LIN {X 0,Y 474.699,Z 220.358,A -85,B 0,C 180,E1 -7395.456,E2 -7395.456} C_VEL
LIN {X 0,Y 474.663,Z 220.354,A -85,B 0,C 180,E1 -7399.011,E2 -7399.011} C_VEL
LIN {X 0,Y 474.589,Z 220.363,A -85,B 0,C 180,E1 -7401.729,E2 -7401.729} C_VEL
LIN {X 0,Y 474.629,Z 220.358,A -85,B 0,C 180,E1 -7404.495,E2 -7404.495} C_VEL
LIN {X 0,Y 474.675,Z 220.357,A -85,B 0,C 180,E1 -7407.333,E2 -7407.333} C_VEL
LIN {X 0,Y 474.605,Z 220.36,A -85,B 0,C 180,E1 -7410.23,E2 -7410.23} C_VEL
LIN {X 0,Y 474.645,Z 220.363,A -85,B 0,C 180,E1 -7413.22,E2 -7413.22} C_VEL
LIN {X 0,Y 474.586,Z 220.363,A -85,B 0,C 180,E1 -7416.324,E2 -7416.324} C_VEL
LIN {X 0,Y 474.615,Z 220.366,A -85,B 0,C 180,E1 -7419.646,E2 -7419.646} C_VEL
LIN {X 0,Y 474.602,Z 220.363,A -85,B 0,C 180,E1 -7422.234,E2 -7422.234} C_VEL
LIN {X 0,Y 474.618,Z 220.369,A -85,B 0,C 180,E1 -7425.298,E2 -7425.298} C_VEL
LIN {X 0,Y 474.617,Z 220.364,A -85,B 0,C 180,E1 -7428.214,E2 -7428.214} C_VEL
LIN {X 0,Y 474.612,Z 220.371,A -85,B 0,C 180,E1 -7431.543,E2 -7431.543} C_VEL
LIN {X 0,Y 474.624,Z 220.364,A -85,B 0,C 180,E1 -7434.726,E2 -7434.726} C_VEL
LIN {X 0,Y 474.638,Z 220.362,A -85,B 0,C 180,E1 -7437.788,E2 -7437.788} C_VEL
LIN {X 0,Y 474.61,Z 220.362,A -85,B 0,C 180,E1 -7440.889,E2 -7440.889} C_VEL
LIN {X 0,Y 474.677,Z 220.486,A -85,B 0,C 180,E1 -7442.491,E2 -7442.491} C_VEL
LIN {X 0,Y 475.888,Z 227.892,A -85,B 0,C 180,E1 -7444.05,E2 -7444.05} C_VEL
LIN {X 0,Y 475.509,Z 242.561,A -85,B 0,C 180,E1 -7446.942,E2 -7446.942} C_VEL
LIN {X 0,Y 475.457,Z 243.986,A -85,B 0,C 180,E1 -7447.219,E2 -7447.219} C_VEL
LIN {X 0,Y 477.495,Z 254.111,A -85,B 0,C 180,E1 -7447.465,E2 -7447.465} C_VEL
LIN {X 0,Y 477.669,Z 257.985,A -85,B 0,C 180,E1 -7447.532,E2 -7447.532} C_VEL
LIN {X 0,Y 477.181,Z 261.87,A -85,B 0,C 180,E1 -7447.573,E2 -7447.573} C_VEL
LIN {X 0,Y 475.045,Z 269.533,A -85,B 0,C 180,E1 -7447.609,E2 -7447.609} C_VEL
LIN {X 0,Y 472.115,Z 279.174,A -85,B 0,C 180,E1 -7447.645,E2 -7447.645} C_VEL
LIN {X 0,Y 471.398,Z 285.1,A -85,B 0,C 180,E1 -7447.71,E2 -7447.71} C_VEL
LIN {X 0,Y 470.736,Z 351.494,A -85,B 0,C 180,E1 -7448.745,E2 -7448.745} C_VEL
LIN {X 0,Y 470.477,Z 364.16,A -85,B 0,C 180,E1 -7449.106,E2 -7449.106} C_VEL
LIN {X 0,Y 470.075,Z 377.21,A -85,B 0,C 180,E1 -7449.659,E2 -7449.659} C_VEL
LIN {X 0,Y 469.661,Z 388.302,A -85,B 0,C 180,E1 -7450.296,E2 -7450.296} C_VEL
LIN {X 0,Y 469.132,Z 400.52,A -85,B 0,C 180,E1 -7451.211,E2 -7451.211} C_VEL
LIN {X 0,Y 468.614,Z 411.084,A -85,B 0,C 180,E1 -7452.207,E2 -7452.207} C_VEL
LIN {X 0,Y 468.122,Z 419.679,A -85,B 0,C 180,E1 -7453.202,E2 -7453.202} C_VEL
LIN {X 0,Y 467.705,Z 427.565,A -85,B 0,C 180,E1 -7454.307,E2 -7454.307} C_VEL
LIN {X 0,Y 467.365,Z 435.229,A -85,B 0,C 180,E1 -7455.634,E2 -7455.634} C_VEL
LIN {X 0,Y 467.136,Z 441.363,A -85,B 0,C 180,E1 -7456.958,E2 -7456.958} C_VEL
LIN {X 0,Y 466.936,Z 446.542,A -85,B 0,C 180,E1 -7458.382,E2 -7458.382} C_VEL
LIN {X 0,Y 466.762,Z 449.893,A -85,B 0,C 180,E1 -7459.59,E2 -7459.59} C_VEL
LIN {X 0,Y 466.642,Z 451.795,A -85,B 0,C 180,E1 -7460.464,E2 -7460.464} C_VEL
LIN {X 0,Y 466.643,Z 453.238,A -85,B 0,C 180,E1 -7461.338,E2 -7461.338} C_VEL
LIN {X 0,Y 466.676,Z 454.878,A -85,B 0,C 180,E1 -7463.08,E2 -7463.08} C_VEL
LIN {X 0,Y 466.646,Z 455.12,A -85,B 0,C 180,E1 -7463.948,E2 -7463.948} C_VEL
LIN {X 0,Y 466.65,Z 454.939,A -85,B 0,C 180,E1 -7464.815,E2 -7464.815} C_VEL
LIN {X 0,Y 466.683,Z 453.385,A -85,B 0,C 180,E1 -7466.547,E2 -7466.547} C_VEL
LIN {X 0,Y 466.706,Z 452.028,A -85,B 0,C 180,E1 -7467.411,E2 -7467.411} C_VEL
LIN {X 0,Y 466.724,Z 449.165,A -85,B 0,C 180,E1 -7468.706,E2 -7468.706} C_VEL
LIN {X 0,Y 466.769,Z 445.291,A -85,B 0,C 180,E1 -7470,E2 -7470} C_VEL
LIN {X 0,Y 467.063,Z 440.289,A -85,B 0,C 180,E1 -7471.293,E2 -7471.293} C_VEL
LIN {X 0,Y 467.253,Z 434.025,A -85,B 0,C 180,E1 -7472.586,E2 -7472.586} C_VEL
LIN {X 0,Y 467.656,Z 426.185,A -85,B 0,C 180,E1 -7473.878,E2 -7473.878} C_VEL
LIN {X 0,Y 468.117,Z 418.205,A -85,B 0,C 180,E1 -7474.952,E2 -7474.952} C_VEL
LIN {X 0,Y 468.566,Z 408.492,A -85,B 0,C 180,E1 -7476.027,E2 -7476.027} C_VEL
LIN {X 0,Y 469.086,Z 397.645,A -85,B 0,C 180,E1 -7476.992,E2 -7476.992} C_VEL
LIN {X 0,Y 469.593,Z 385.29,A -85,B 0,C 180,E1 -7477.849,E2 -7477.849} C_VEL
LIN {X 0,Y 470.024,Z 373.161,A -85,B 0,C 180,E1 -7478.491,E2 -7478.491} C_VEL
LIN {X 0,Y 470.342,Z 360.402,A -85,B 0,C 180,E1 -7478.972,E2 -7478.972} C_VEL
LIN {X 0,Y 470.527,Z 346.91,A -85,B 0,C 180,E1 -7479.294,E2 -7479.294} C_VEL
LIN {X 0,Y 471.18,Z 259.024,A -85,B 0,C 180,E1 -7480.637,E2 -7480.637} C_VEL
LIN {X 0,Y 468.414,Z 244.125,A -85,B 0,C 180,E1 -7480.974,E2 -7480.974} C_VEL
LIN {X 0,Y 468.806,Z 229.463,A -85,B 0,C 180,E1 -7483.878,E2 -7483.878} C_VEL
LIN {X 0,Y 468.381,Z 225.11,A -85,B 0,C 180,E1 -7484.778,E2 -7484.778} C_VEL
LIN {X 0,Y 467.657,Z 221.233,A -85,B 0,C 180,E1 -7485.638,E2 -7485.638} C_VEL
LIN {X 0,Y 467.617,Z 221.24,A -85,B 0,C 180,E1 -7488.763,E2 -7488.763} C_VEL
LIN {X 0,Y 467.584,Z 221.237,A -85,B 0,C 180,E1 -7491.268,E2 -7491.268} C_VEL
LIN {X 0,Y 467.566,Z 221.238,A -85,B 0,C 180,E1 -7493.944,E2 -7493.944} C_VEL
LIN {X 0,Y 467.568,Z 221.245,A -85,B 0,C 180,E1 -7496.803,E2 -7496.803} C_VEL
LIN {X 0,Y 467.55,Z 221.24,A -85,B 0,C 180,E1 -7499.738,E2 -7499.738} C_VEL
LIN {X 0,Y 467.586,Z 221.243,A -85,B 0,C 180,E1 -7502.758,E2 -7502.758} C_VEL
LIN {X 0,Y 467.555,Z 221.24,A -85,B 0,C 180,E1 -7505.889,E2 -7505.889} C_VEL
LIN {X 0,Y 467.577,Z 221.239,A -85,B 0,C 180,E1 -7509.145,E2 -7509.145} C_VEL
LIN {X 0,Y 467.588,Z 221.242,A -85,B 0,C 180,E1 -7512.567,E2 -7512.567} C_VEL
LIN {X 0,Y 467.567,Z 221.241,A -85,B 0,C 180,E1 -7515.052,E2 -7515.052} C_VEL
LIN {X 0,Y 467.575,Z 221.245,A -85,B 0,C 180,E1 -7518.596,E2 -7518.596} C_VEL
LIN {X 0,Y 467.56,Z 221.239,A -85,B 0,C 180,E1 -7521.409,E2 -7521.409} C_VEL
LIN {X 0,Y 467.559,Z 221.242,A -85,B 0,C 180,E1 -7524.261,E2 -7524.261} C_VEL
LIN {X 0,Y 467.583,Z 221.237,A -85,B 0,C 180,E1 -7527.321,E2 -7527.321} C_VEL
LIN {X 0,Y 467.57,Z 221.246,A -85,B 0,C 180,E1 -7530.667,E2 -7530.667} C_VEL
LIN {X 0,Y 467.587,Z 221.237,A -85,B 0,C 180,E1 -7533.198,E2 -7533.198} C_VEL
LIN {X 0,Y 467.59,Z 221.241,A -85,B 0,C 180,E1 -7536.469,E2 -7536.469} C_VEL
LIN {X 0,Y 467.623,Z 221.231,A -85,B 0,C 180,E1 -7539.777,E2 -7539.777} C_VEL
LIN {X 0,Y 467.596,Z 221.241,A -85,B 0,C 180,E1 -7542.506,E2 -7542.506} C_VEL
LIN {X 0,Y 467.602,Z 221.235,A -85,B 0,C 180,E1 -7545.196,E2 -7545.196} C_VEL
LIN {X 0,Y 467.657,Z 221.227,A -85,B 0,C 180,E1 -7547.854,E2 -7547.854} C_VEL
LIN {X 0,Y 467.67,Z 221.226,A -85,B 0,C 180,E1 -7551.357,E2 -7551.357} C_VEL
LIN {X 0,Y 467.724,Z 221.219,A -85,B 0,C 180,E1 -7553.962,E2 -7553.962} C_VEL
LIN {X 0,Y 467.859,Z 221.202,A -85,B 0,C 180,E1 -7557.417,E2 -7557.417} C_VEL
LIN {X 0,Y 467.882,Z 221.2,A -85,B 0,C 180,E1 -7560,E2 -7560} C_VEL
LIN {X 0,Y 467.852,Z 221.211,A -85,B 0,C 180,E1 -7562.583,E2 -7562.583} C_VEL
LIN {X 0,Y 467.743,Z 221.218,A -85,B 0,C 180,E1 -7566.037,E2 -7566.037} C_VEL
LIN {X 0,Y 467.68,Z 221.232,A -85,B 0,C 180,E1 -7568.643,E2 -7568.643} C_VEL
LIN {X 0,Y 467.657,Z 221.229,A -85,B 0,C 180,E1 -7572.145,E2 -7572.145} C_VEL
LIN {X 0,Y 467.64,Z 221.229,A -85,B 0,C 180,E1 -7575.695,E2 -7575.695} C_VEL
LIN {X 0,Y 467.622,Z 221.232,A -85,B 0,C 180,E1 -7579.308,E2 -7579.308} C_VEL
LIN {X 0,Y 467.535,Z 221.244,A -85,B 0,C 180,E1 -7582.074,E2 -7582.074} C_VEL
LIN {X 0,Y 467.586,Z 221.24,A -85,B 0,C 180,E1 -7584.888,E2 -7584.888} C_VEL
LIN {X 0,Y 467.58,Z 221.237,A -85,B 0,C 180,E1 -7587.772,E2 -7587.772} C_VEL
LIN {X 0,Y 467.569,Z 221.24,A -85,B 0,C 180,E1 -7591.045,E2 -7591.045} C_VEL
LIN {X 0,Y 467.577,Z 221.241,A -85,B 0,C 180,E1 -7594.24,E2 -7594.24} C_VEL
LIN {X 0,Y 467.543,Z 221.242,A -85,B 0,C 180,E1 -7597.186,E2 -7597.186} C_VEL
LIN {X 0,Y 467.57,Z 221.242,A -85,B 0,C 180,E1 -7600.265,E2 -7600.265} C_VEL
LIN {X 0,Y 467.56,Z 221.247,A -85,B 0,C 180,E1 -7602.563,E2 -7602.563} C_VEL
LIN {X 0,Y 467.566,Z 221.24,A -85,B 0,C 180,E1 -7605.053,E2 -7605.053} C_VEL
LIN {X 0,Y 467.574,Z 221.245,A -85,B 0,C 180,E1 -7608.597,E2 -7608.597} C_VEL
LIN {X 0,Y 467.559,Z 221.239,A -85,B 0,C 180,E1 -7611.41,E2 -7611.41} C_VEL
LIN {X 0,Y 467.559,Z 221.244,A -85,B 0,C 180,E1 -7614.261,E2 -7614.261} C_VEL
LIN {X 0,Y 467.583,Z 221.236,A -85,B 0,C 180,E1 -7617.321,E2 -7617.321} C_VEL
LIN {X 0,Y 467.57,Z 221.245,A -85,B 0,C 180,E1 -7620.668,E2 -7620.668} C_VEL
LIN {X 0,Y 467.588,Z 221.241,A -85,B 0,C 180,E1 -7623.198,E2 -7623.198} C_VEL
LIN {X 0,Y 467.635,Z 221.409,A -85,B 0,C 180,E1 -7624.591,E2 -7624.591} C_VEL
LIN {X 0,Y 469.581,Z 232.099,A -85,B 0,C 180,E1 -7626.633,E2 -7626.633} C_VEL
LIN {X 0,Y 469.081,Z 247.517,A -85,B 0,C 180,E1 -7629.385,E2 -7629.385} C_VEL
LIN {X 0,Y 468.359,Z 265.424,A -85,B 0,C 180,E1 -7632.536,E2 -7632.536} C_VEL
LIN {X 0,Y 468.254,Z 268.418,A -85,B 0,C 180,E1 -7633.06,E2 -7633.06} C_VEL
LIN {X 0,Y 471.044,Z 286.992,A -85,B 0,C 180,E1 -7633.443,E2 -7633.443} C_VEL
LIN {X 0,Y 470.421,Z 377.296,A -85,B 0,C 180,E1 -7634.844,E2 -7634.844} C_VEL
LIN {X 0,Y 470.028,Z 390.369,A -85,B 0,C 180,E1 -7635.219,E2 -7635.219} C_VEL
LIN {X 0,Y 469.581,Z 403.006,A -85,B 0,C 180,E1 -7635.758,E2 -7635.758} C_VEL
LIN {X 0,Y 469.116,Z 415.032,A -85,B 0,C 180,E1 -7636.462,E2 -7636.462} C_VEL
LIN {X 0,Y 468.598,Z 426.01,A -85,B 0,C 180,E1 -7637.285,E2 -7637.285} C_VEL
LIN {X 0,Y 468.165,Z 436.903,A -85,B 0,C 180,E1 -7638.308,E2 -7638.308} C_VEL
LIN {X 0,Y 467.712,Z 446.199,A -85,B 0,C 180,E1 -7639.393,E2 -7639.393} C_VEL
LIN {X 0,Y 467.29,Z 455.223,A -85,B 0,C 180,E1 -7640.696,E2 -7640.696} C_VEL
LIN {X 0,Y 467.012,Z 462.49,A -85,B 0,C 180,E1 -7641.998,E2 -7641.998} C_VEL
LIN {X 0,Y 466.852,Z 467.395,A -85,B 0,C 180,E1 -7643.083,E2 -7643.083} C_VEL
LIN {X 0,Y 466.76,Z 472.159,A -85,B 0,C 180,E1 -7644.383,E2 -7644.383} C_VEL
LIN {X 0,Y 466.646,Z 475.799,A -85,B 0,C 180,E1 -7645.681,E2 -7645.681} C_VEL
LIN {X 0,Y 466.689,Z 477.682,A -85,B 0,C 180,E1 -7646.547,E2 -7646.547} C_VEL
LIN {X 0,Y 466.662,Z 479.097,A -85,B 0,C 180,E1 -7647.411,E2 -7647.411} C_VEL
LIN {X 0,Y 466.619,Z 480.721,A -85,B 0,C 180,E1 -7649.137,E2 -7649.137} C_VEL
LIN {X 0,Y 466.6,Z 480.951,A -85,B 0,C 180,E1 -7650,E2 -7650} C_VEL
LIN {X 0,Y 466.619,Z 480.752,A -85,B 0,C 180,E1 -7650.863,E2 -7650.863} C_VEL
LIN {X 0,Y 466.662,Z 479.171,A -85,B 0,C 180,E1 -7652.59,E2 -7652.59} C_VEL
LIN {X 0,Y 466.688,Z 477.792,A -85,B 0,C 180,E1 -7653.453,E2 -7653.453} C_VEL
LIN {X 0,Y 466.688,Z 474.878,A -85,B 0,C 180,E1 -7654.751,E2 -7654.751} C_VEL
LIN {X 0,Y 466.75,Z 470.937,A -85,B 0,C 180,E1 -7656.05,E2 -7656.05} C_VEL
LIN {X 0,Y 466.936,Z 465.869,A -85,B 0,C 180,E1 -7657.35,E2 -7657.35} C_VEL
LIN {X 0,Y 467.163,Z 459.502,A -85,B 0,C 180,E1 -7658.652,E2 -7658.652} C_VEL
LIN {X 0,Y 467.528,Z 451.545,A -85,B 0,C 180,E1 -7659.955,E2 -7659.955} C_VEL
LIN {X 0,Y 467.928,Z 443.451,A -85,B 0,C 180,E1 -7661.04,E2 -7661.04} C_VEL
LIN {X 0,Y 468.467,Z 433.592,A -85,B 0,C 180,E1 -7662.124,E2 -7662.124} C_VEL
LIN {X 0,Y 468.907,Z 422.696,A -85,B 0,C 180,E1 -7663.091,E2 -7663.091} C_VEL
LIN {X 0,Y 469.455,Z 411.742,A -85,B 0,C 180,E1 -7663.859,E2 -7663.859} C_VEL
LIN {X 0,Y 469.955,Z 399.836,A -85,B 0,C 180,E1 -7664.507,E2 -7664.507} C_VEL
LIN {X 0,Y 470.414,Z 386.948,A -85,B 0,C 180,E1 -7665.018,E2 -7665.018} C_VEL
LIN {X 0,Y 470.738,Z 374.239,A -85,B 0,C 180,E1 -7665.339,E2 -7665.339} C_VEL
LIN {X 0,Y 471.322,Z 286.387,A -85,B 0,C 180,E1 -7666.703,E2 -7666.703} C_VEL
LIN {X 0,Y 468.345,Z 268.311,A -85,B 0,C 180,E1 -7667.111,E2 -7667.111} C_VEL
LIN {X 0,Y 469.121,Z 251.176,A -85,B 0,C 180,E1 -7670.155,E2 -7670.155} C_VEL
LIN {X 0,Y 469.854,Z 234.766,A -85,B 0,C 180,E1 -7673.119,E2 -7673.119} C_VEL
LIN {X 0,Y 469.386,Z 229.989,A -85,B 0,C 180,E1 -7674.029,E2 -7674.029} C_VEL
LIN {X 0,Y 467.588,Z 221.245,A -85,B 0,C 180,E1 -7675.801,E2 -7675.801} C_VEL
LIN {X 0,Y 467.558,Z 221.246,A -85,B 0,C 180,E1 -7678.751,E2 -7678.751} C_VEL
LIN {X 0,Y 467.584,Z 221.242,A -85,B 0,C 180,E1 -7681.74,E2 -7681.74} C_VEL
LIN {X 0,Y 467.564,Z 221.241,A -85,B 0,C 180,E1 -7684.833,E2 -7684.833} C_VEL
LIN {X 0,Y 467.563,Z 221.241,A -85,B 0,C 180,E1 -7688.045,E2 -7688.045} C_VEL
LIN {X 0,Y 467.576,Z 221.244,A -85,B 0,C 180,E1 -7691.276,E2 -7691.276} C_VEL
LIN {X 0,Y 467.547,Z 221.245,A -85,B 0,C 180,E1 -7693.82,E2 -7693.82} C_VEL
LIN {X 0,Y 467.549,Z 221.242,A -85,B 0,C 180,E1 -7696.255,E2 -7696.255} C_VEL
LIN {X 0,Y 467.575,Z 221.239,A -85,B 0,C 180,E1 -7698.724,E2 -7698.724} C_VEL
LIN {X 0,Y 467.562,Z 221.24,A -85,B 0,C 180,E1 -7701.955,E2 -7701.955} C_VEL
LIN {X 0,Y 467.557,Z 221.244,A -85,B 0,C 180,E1 -7705.167,E2 -7705.167} C_VEL
LIN {X 0,Y 467.583,Z 221.237,A -85,B 0,C 180,E1 -7708.26,E2 -7708.26} C_VEL
LIN {X 0,Y 467.556,Z 221.241,A -85,B 0,C 180,E1 -7711.249,E2 -7711.249} C_VEL
LIN {X 0,Y 467.585,Z 221.233,A -85,B 0,C 180,E1 -7714.159,E2 -7714.159} C_VEL
LIN {X 0,Y 467.577,Z 221.24,A -85,B 0,C 180,E1 -7716.996,E2 -7716.996} C_VEL
LIN {X 0,Y 467.623,Z 221.235,A -85,B 0,C 180,E1 -7719.777,E2 -7719.777} C_VEL
LIN {X 0,Y 467.599,Z 221.233,A -85,B 0,C 180,E1 -7722.506,E2 -7722.506} C_VEL
LIN {X 0,Y 467.61,Z 221.237,A -85,B 0,C 180,E1 -7725.197,E2 -7725.197} C_VEL
LIN {X 0,Y 467.657,Z 221.226,A -85,B 0,C 180,E1 -7727.855,E2 -7727.855} C_VEL
LIN {X 0,Y 467.681,Z 221.231,A -85,B 0,C 180,E1 -7731.357,E2 -7731.357} C_VEL
LIN {X 0,Y 467.743,Z 221.217,A -85,B 0,C 180,E1 -7733.963,E2 -7733.963} C_VEL
LIN {X 0,Y 467.849,Z 221.206,A -85,B 0,C 180,E1 -7737.417,E2 -7737.417} C_VEL
LIN {X 0,Y 467.882,Z 221.201,A -85,B 0,C 180,E1 -7740,E2 -7740} C_VEL
LIN {X 0,Y 467.852,Z 221.2,A -85,B 0,C 180,E1 -7742.583,E2 -7742.583} C_VEL
LIN {X 0,Y 467.724,Z 221.22,A -85,B 0,C 180,E1 -7746.038,E2 -7746.038} C_VEL
LIN {X 0,Y 467.67,Z 221.221,A -85,B 0,C 180,E1 -7748.643,E2 -7748.643} C_VEL
LIN {X 0,Y 467.657,Z 221.226,A -85,B 0,C 180,E1 -7752.146,E2 -7752.146} C_VEL
LIN {X 0,Y 467.639,Z 221.233,A -85,B 0,C 180,E1 -7755.695,E2 -7755.695} C_VEL
LIN {X 0,Y 467.622,Z 221.234,A -85,B 0,C 180,E1 -7759.308,E2 -7759.308} C_VEL
LIN {X 0,Y 467.535,Z 221.239,A -85,B 0,C 180,E1 -7762.074,E2 -7762.074} C_VEL
LIN {X 0,Y 467.57,Z 221.24,A -85,B 0,C 180,E1 -7764.889,E2 -7764.889} C_VEL
LIN {X 0,Y 467.617,Z 221.236,A -85,B 0,C 180,E1 -7767.769,E2 -7767.769} C_VEL
LIN {X 0,Y 467.569,Z 221.24,A -85,B 0,C 180,E1 -7771.045,E2 -7771.045} C_VEL
LIN {X 0,Y 467.589,Z 221.236,A -85,B 0,C 180,E1 -7774.242,E2 -7774.242} C_VEL
LIN {X 0,Y 467.544,Z 221.245,A -85,B 0,C 180,E1 -7777.186,E2 -7777.186} C_VEL
LIN {X 0,Y 467.574,Z 221.238,A -85,B 0,C 180,E1 -7780.265,E2 -7780.265} C_VEL
LIN {X 0,Y 467.55,Z 221.246,A -85,B 0,C 180,E1 -7783.745,E2 -7783.745} C_VEL
LIN {X 0,Y 467.55,Z 221.239,A -85,B 0,C 180,E1 -7786.255,E2 -7786.255} C_VEL
LIN {X 0,Y 467.577,Z 221.242,A -85,B 0,C 180,E1 -7788.724,E2 -7788.724} C_VEL
LIN {X 0,Y 467.566,Z 221.244,A -85,B 0,C 180,E1 -7791.956,E2 -7791.956} C_VEL
LIN {X 0,Y 467.561,Z 221.247,A -85,B 0,C 180,E1 -7795.167,E2 -7795.167} C_VEL
LIN {X 0,Y 467.585,Z 221.237,A -85,B 0,C 180,E1 -7798.26,E2 -7798.26} C_VEL
LIN {X 0,Y 467.561,Z 221.24,A -85,B 0,C 180,E1 -7801.249,E2 -7801.249} C_VEL
LIN {X 0,Y 467.642,Z 221.348,A -85,B 0,C 180,E1 -7802.279,E2 -7802.279} C_VEL
LIN {X 0,Y 468.846,Z 228.085,A -85,B 0,C 180,E1 -7803.723,E2 -7803.723} C_VEL
LIN {X 0,Y 468.702,Z 240.004,A -85,B 0,C 180,E1 -7806.118,E2 -7806.118} C_VEL
LIN {X 0,Y 468.586,Z 244.465,A -85,B 0,C 180,E1 -7806.954,E2 -7806.954} C_VEL
LIN {X 0,Y 471.64,Z 260.33,A -85,B 0,C 180,E1 -7807.33,E2 -7807.33} C_VEL
LIN {X 0,Y 471.398,Z 285.1,A -85,B 0,C 180,E1 -7807.71,E2 -7807.71} C_VEL
LIN {X 0,Y 470.73,Z 290.948,A -85,B 0,C 180,E1 -7807.775,E2 -7807.775} C_VEL
LIN {X 0,Y 465.011,Z 309.952,A -85,B 0,C 180,E1 -7807.85,E2 -7807.85} C_VEL
LIN {X 0,Y 464.34,Z 315.8,A -85,B 0,C 180,E1 -7807.916,E2 -7807.916} C_VEL
LIN {X 0,Y 463.955,Z 352.222,A -85,B 0,C 180,E1 -7808.507,E2 -7808.507} C_VEL
LIN {X 0,Y 463.666,Z 364.704,A -85,B 0,C 180,E1 -7808.871,E2 -7808.871} C_VEL
LIN {X 0,Y 463.282,Z 377.09,A -85,B 0,C 180,E1 -7809.405,E2 -7809.405} C_VEL
LIN {X 0,Y 462.816,Z 388.516,A -85,B 0,C 180,E1 -7810.068,E2 -7810.068} C_VEL
LIN {X 0,Y 462.286,Z 399.871,A -85,B 0,C 180,E1 -7810.922,E2 -7810.922} C_VEL
LIN {X 0,Y 461.731,Z 410.578,A -85,B 0,C 180,E1 -7811.933,E2 -7811.933} C_VEL
LIN {X 0,Y 461.198,Z 419.289,A -85,B 0,C 180,E1 -7812.942,E2 -7812.942} C_VEL
LIN {X 0,Y 460.779,Z 427.286,A -85,B 0,C 180,E1 -7814.065,E2 -7814.065} C_VEL
LIN {X 0,Y 460.398,Z 435.056,A -85,B 0,C 180,E1 -7815.412,E2 -7815.412} C_VEL
LIN {X 0,Y 460.092,Z 441.258,A -85,B 0,C 180,E1 -7816.754,E2 -7816.754} C_VEL
LIN {X 0,Y 459.878,Z 445.793,A -85,B 0,C 180,E1 -7817.98,E2 -7817.98} C_VEL
LIN {X 0,Y 459.703,Z 449.912,A -85,B 0,C 180,E1 -7819.429,E2 -7819.429} C_VEL
LIN {X 0,Y 459.563,Z 451.842,A -85,B 0,C 180,E1 -7820.316,E2 -7820.316} C_VEL
LIN {X 0,Y 459.544,Z 453.34,A -85,B 0,C 180,E1 -7821.203,E2 -7821.203} C_VEL
LIN {X 0,Y 459.572,Z 455.035,A -85,B 0,C 180,E1 -7822.973,E2 -7822.973} C_VEL
LIN {X 0,Y 459.592,Z 455.303,A -85,B 0,C 180,E1 -7823.855,E2 -7823.855} C_VEL
LIN {X 0,Y 459.56,Z 455.174,A -85,B 0,C 180,E1 -7824.735,E2 -7824.735} C_VEL
LIN {X 0,Y 459.578,Z 453.675,A -85,B 0,C 180,E1 -7826.493,E2 -7826.493} C_VEL
LIN {X 0,Y 459.624,Z 452.344,A -85,B 0,C 180,E1 -7827.371,E2 -7827.371} C_VEL
LIN {X 0,Y 459.648,Z 449.537,A -85,B 0,C 180,E1 -7828.686,E2 -7828.686} C_VEL
LIN {X 0,Y 459.691,Z 445.722,A -85,B 0,C 180,E1 -7830,E2 -7830} C_VEL
LIN {X 0,Y 459.971,Z 440.784,A -85,B 0,C 180,E1 -7831.313,E2 -7831.313} C_VEL
LIN {X 0,Y 460.185,Z 434.599,A -85,B 0,C 180,E1 -7832.626,E2 -7832.626} C_VEL
LIN {X 0,Y 460.476,Z 428.278,A -85,B 0,C 180,E1 -7833.719,E2 -7833.719} C_VEL
LIN {X 0,Y 460.952,Z 420.692,A -85,B 0,C 180,E1 -7834.81,E2 -7834.81} C_VEL
LIN {X 0,Y 461.485,Z 411.491,A -85,B 0,C 180,E1 -7835.9,E2 -7835.9} C_VEL
LIN {X 0,Y 461.997,Z 401.266,A -85,B 0,C 180,E1 -7836.88,E2 -7836.88} C_VEL
LIN {X 0,Y 462.505,Z 389.939,A -85,B 0,C 180,E1 -7837.751,E2 -7837.751} C_VEL
LIN {X 0,Y 462.966,Z 378.139,A -85,B 0,C 180,E1 -7838.457,E2 -7838.457} C_VEL
LIN {X 0,Y 463.333,Z 365.061,A -85,B 0,C 180,E1 -7839.027,E2 -7839.027} C_VEL
LIN {X 0,Y 463.601,Z 352.075,A -85,B 0,C 180,E1 -7839.407,E2 -7839.407} C_VEL
LIN {X 0,Y 464.359,Z 260.187,A -85,B 0,C 180,E1 -7840.85,E2 -7840.85} C_VEL
LIN {X 0,Y 461.455,Z 244.238,A -85,B 0,C 180,E1 -7841.225,E2 -7841.225} C_VEL
LIN {X 0,Y 461.845,Z 229.938,A -85,B 0,C 180,E1 -7844.092,E2 -7844.092} C_VEL
LIN {X 0,Y 460.607,Z 222.112,A -85,B 0,C 180,E1 -7845.791,E2 -7845.791} C_VEL
LIN {X 0,Y 460.571,Z 222.116,A -85,B 0,C 180,E1 -7848.9,E2 -7848.9} C_VEL
LIN {X 0,Y 460.519,Z 222.116,A -85,B 0,C 180,E1 -7851.485,E2 -7851.485} C_VEL
LIN {X 0,Y 460.534,Z 222.118,A -85,B 0,C 180,E1 -7854.333,E2 -7854.333} C_VEL
LIN {X 0,Y 460.537,Z 222.115,A -85,B 0,C 180,E1 -7857.246,E2 -7857.246} C_VEL
LIN {X 0,Y 460.511,Z 222.12,A -85,B 0,C 180,E1 -7860.24,E2 -7860.24} C_VEL
LIN {X 0,Y 460.531,Z 222.115,A -85,B 0,C 180,E1 -7863.325,E2 -7863.325} C_VEL
LIN {X 0,Y 460.478,Z 222.127,A -85,B 0,C 180,E1 -7866.529,E2 -7866.529} C_VEL
LIN {X 0,Y 460.529,Z 222.115,A -85,B 0,C 180,E1 -7869.863,E2 -7869.863} C_VEL
LIN {X 0,Y 460.515,Z 222.122,A -85,B 0,C 180,E1 -7872.9,E2 -7872.9} C_VEL
LIN {X 0,Y 460.507,Z 222.118,A -85,B 0,C 180,E1 -7875.831,E2 -7875.831} C_VEL
LIN {X 0,Y 460.529,Z 222.119,A -85,B 0,C 180,E1 -7878.988,E2 -7878.988} C_VEL
LIN {X 0,Y 460.523,Z 222.117,A -85,B 0,C 180,E1 -7881.266,E2 -7881.266} C_VEL
LIN {X 0,Y 460.51,Z 222.124,A -85,B 0,C 180,E1 -7884.554,E2 -7884.554} C_VEL
LIN {X 0,Y 460.533,Z 222.114,A -85,B 0,C 180,E1 -7887.715,E2 -7887.715} C_VEL
LIN {X 0,Y 460.54,Z 222.12,A -85,B 0,C 180,E1 -7890.769,E2 -7890.769} C_VEL
LIN {X 0,Y 460.542,Z 222.113,A -85,B 0,C 180,E1 -7893.733,E2 -7893.733} C_VEL
LIN {X 0,Y 460.544,Z 222.121,A -85,B 0,C 180,E1 -7896.624,E2 -7896.624} C_VEL
LIN {X 0,Y 460.552,Z 222.112,A -85,B 0,C 180,E1 -7899.453,E2 -7899.453} C_VEL
LIN {X 0,Y 460.548,Z 222.115,A -85,B 0,C 180,E1 -7902.23,E2 -7902.23} C_VEL
LIN {X 0,Y 460.562,Z 222.114,A -85,B 0,C 180,E1 -7904.965,E2 -7904.965} C_VEL
LIN {X 0,Y 460.61,Z 222.105,A -85,B 0,C 180,E1 -7907.666,E2 -7907.666} C_VEL
LIN {X 0,Y 460.62,Z 222.105,A -85,B 0,C 180,E1 -7911.224,E2 -7911.224} C_VEL
LIN {X 0,Y 460.688,Z 222.095,A -85,B 0,C 180,E1 -7913.87,E2 -7913.87} C_VEL
LIN {X 0,Y 460.8,Z 222.081,A -85,B 0,C 180,E1 -7917.377,E2 -7917.377} C_VEL
LIN {X 0,Y 460.852,Z 222.076,A -85,B 0,C 180,E1 -7920,E2 -7920} C_VEL
LIN {X 0,Y 460.793,Z 222.09,A -85,B 0,C 180,E1 -7922.622,E2 -7922.622} C_VEL
LIN {X 0,Y 460.709,Z 222.095,A -85,B 0,C 180,E1 -7926.13,E2 -7926.13} C_VEL
LIN {X 0,Y 460.627,Z 222.108,A -85,B 0,C 180,E1 -7928.776,E2 -7928.776} C_VEL
LIN {X 0,Y 460.614,Z 222.11,A -85,B 0,C 180,E1 -7932.445,E2 -7932.445} C_VEL
LIN {X 0,Y 460.601,Z 222.107,A -85,B 0,C 180,E1 -7935.997,E2 -7935.997} C_VEL
LIN {X 0,Y 460.569,Z 222.11,A -85,B 0,C 180,E1 -7939.616,E2 -7939.616} C_VEL
LIN {X 0,Y 460.511,Z 222.123,A -85,B 0,C 180,E1 -7942.429,E2 -7942.429} C_VEL
LIN {X 0,Y 460.549,Z 222.113,A -85,B 0,C 180,E1 -7945.797,E2 -7945.797} C_VEL
LIN {X 0,Y 460.527,Z 222.119,A -85,B 0,C 180,E1 -7948.235,E2 -7948.235} C_VEL
LIN {X 0,Y 460.521,Z 222.116,A -85,B 0,C 180,E1 -7951.283,E2 -7951.283} C_VEL
LIN {X 0,Y 460.523,Z 222.123,A -85,B 0,C 180,E1 -7954.504,E2 -7954.504} C_VEL
LIN {X 0,Y 460.499,Z 222.118,A -85,B 0,C 180,E1 -7957.623,E2 -7957.623} C_VEL
LIN {X 0,Y 460.527,Z 222.117,A -85,B 0,C 180,E1 -7961.012,E2 -7961.012} C_VEL
LIN {X 0,Y 460.512,Z 222.125,A -85,B 0,C 180,E1 -7964.589,E2 -7964.589} C_VEL
LIN {X 0,Y 460.504,Z 222.118,A -85,B 0,C 180,E1 -7967.817,E2 -7967.817} C_VEL
LIN {X 0,Y 460.523,Z 222.118,A -85,B 0,C 180,E1 -7970.137,E2 -7970.137} C_VEL
LIN {X 0,Y 460.474,Z 222.122,A -85,B 0,C 180,E1 -7973.47,E2 -7973.47} C_VEL
LIN {X 0,Y 460.53,Z 222.121,A -85,B 0,C 180,E1 -7976.675,E2 -7976.675} C_VEL
LIN {X 0,Y 460.511,Z 222.117,A -85,B 0,C 180,E1 -7979.76,E2 -7979.76} C_VEL
LIN {X 0,Y 460.559,Z 222.118,A -85,B 0,C 180,E1 -7982.755,E2 -7982.755} C_VEL
LIN {X 0,Y 460.552,Z 222.187,A -85,B 0,C 180,E1 -7984.387,E2 -7984.387} C_VEL
LIN {X 0,Y 462.597,Z 233.09,A -85,B 0,C 180,E1 -7986.507,E2 -7986.507} C_VEL
LIN {X 0,Y 462.231,Z 244.609,A -85,B 0,C 180,E1 -7988.598,E2 -7988.598} C_VEL
LIN {X 0,Y 461.52,Z 261.258,A -85,B 0,C 180,E1 -7991.58,E2 -7991.58} C_VEL
LIN {X 0,Y 461.265,Z 268.215,A -85,B 0,C 180,E1 -7992.818,E2 -7992.818} C_VEL
LIN {X 0,Y 464.179,Z 287.594,A -85,B 0,C 180,E1 -7993.225,E2 -7993.225} C_VEL
LIN {X 0,Y 463.562,Z 376.224,A -85,B 0,C 180,E1 -7994.614,E2 -7994.614} C_VEL
LIN {X 0,Y 463.189,Z 388.829,A -85,B 0,C 180,E1 -7994.968,E2 -7994.968} C_VEL
LIN {X 0,Y 462.669,Z 402.385,A -85,B 0,C 180,E1 -7995.541,E2 -7995.541} C_VEL
LIN {X 0,Y 462.181,Z 414.54,A -85,B 0,C 180,E1 -7996.255,E2 -7996.255} C_VEL
LIN {X 0,Y 461.577,Z 426.692,A -85,B 0,C 180,E1 -7997.184,E2 -7997.184} C_VEL
LIN {X 0,Y 461.191,Z 436.517,A -85,B 0,C 180,E1 -7998.128,E2 -7998.128} C_VEL
LIN {X 0,Y 460.672,Z 445.858,A -85,B 0,C 180,E1 -7999.229,E2 -7999.229} C_VEL
LIN {X 0,Y 460.236,Z 454.909,A -85,B 0,C 180,E1 -8000.552,E2 -8000.552} C_VEL
LIN {X 0,Y 459.953,Z 462.199,A -85,B 0,C 180,E1 -8001.875,E2 -8001.875} C_VEL
LIN {X 0,Y 459.743,Z 468.318,A -85,B 0,C 180,E1 -8003.273,E2 -8003.273} C_VEL
LIN {X 0,Y 459.65,Z 473.242,A -85,B 0,C 180,E1 -8004.736,E2 -8004.736} C_VEL
LIN {X 0,Y 459.563,Z 475.56,A -85,B 0,C 180,E1 -8005.615,E2 -8005.615} C_VEL
LIN {X 0,Y 459.584,Z 477.451,A -85,B 0,C 180,E1 -8006.493,E2 -8006.493} C_VEL
LIN {X 0,Y 459.584,Z 478.879,A -85,B 0,C 180,E1 -8007.371,E2 -8007.371} C_VEL
LIN {X 0,Y 459.522,Z 480.515,A -85,B 0,C 180,E1 -8009.124,E2 -8009.124} C_VEL
LIN {X 0,Y 459.531,Z 480.754,A -85,B 0,C 180,E1 -8010,E2 -8010} C_VEL
LIN {X 0,Y 459.522,Z 480.565,A -85,B 0,C 180,E1 -8010.876,E2 -8010.876} C_VEL
LIN {X 0,Y 459.584,Z 478.997,A -85,B 0,C 180,E1 -8012.629,E2 -8012.629} C_VEL
LIN {X 0,Y 459.583,Z 477.624,A -85,B 0,C 180,E1 -8013.507,E2 -8013.507} C_VEL
LIN {X 0,Y 459.616,Z 474.724,A -85,B 0,C 180,E1 -8014.824,E2 -8014.824} C_VEL
LIN {X 0,Y 459.713,Z 469.797,A -85,B 0,C 180,E1 -8016.43,E2 -8016.43} C_VEL
LIN {X 0,Y 459.921,Z 463.766,A -85,B 0,C 180,E1 -8017.905,E2 -8017.905} C_VEL
LIN {X 0,Y 460.22,Z 456.943,A -85,B 0,C 180,E1 -8019.227,E2 -8019.227} C_VEL
LIN {X 0,Y 460.618,Z 448.452,A -85,B 0,C 180,E1 -8020.55,E2 -8020.55} C_VEL
LIN {X 0,Y 461.207,Z 439.732,A -85,B 0,C 180,E1 -8021.649,E2 -8021.649} C_VEL
LIN {X 0,Y 461.75,Z 430.055,A -85,B 0,C 180,E1 -8022.65,E2 -8022.65} C_VEL
LIN {X 0,Y 462.137,Z 419.775,A -85,B 0,C 180,E1 -8023.522,E2 -8023.522} C_VEL
LIN {X 0,Y 462.744,Z 408.345,A -85,B 0,C 180,E1 -8024.288,E2 -8024.288} C_VEL
LIN {X 0,Y 463.249,Z 396.536,A -85,B 0,C 180,E1 -8024.89,E2 -8024.89} C_VEL
LIN {X 0,Y 463.708,Z 383.83,A -85,B 0,C 180,E1 -8025.353,E2 -8025.353} C_VEL
LIN {X 0,Y 463.983,Z 370.733,A -85,B 0,C 180,E1 -8025.653,E2 -8025.653} C_VEL
LIN {X 0,Y 464.618,Z 287.643,A -85,B 0,C 180,E1 -8026.952,E2 -8026.952} C_VEL
LIN {X 0,Y 461.425,Z 268.075,A -85,B 0,C 180,E1 -8027.406,E2 -8027.406} C_VEL
LIN {X 0,Y 462.253,Z 249.857,A -85,B 0,C 180,E1 -8030.701,E2 -8030.701} C_VEL
LIN {X 0,Y 462.939,Z 235.982,A -85,B 0,C 180,E1 -8033.248,E2 -8033.248} C_VEL
LIN {X 0,Y 462.373,Z 230.934,A -85,B 0,C 180,E1 -8034.23,E2 -8034.23} C_VEL
LIN {X 0,Y 460.527,Z 222.124,A -85,B 0,C 180,E1 -8036.058,E2 -8036.058} C_VEL
LIN {X 0,Y 460.528,Z 222.121,A -85,B 0,C 180,E1 -8038.235,E2 -8038.235} C_VEL
LIN {X 0,Y 460.522,Z 222.123,A -85,B 0,C 180,E1 -8041.283,E2 -8041.283} C_VEL
LIN {X 0,Y 460.532,Z 222.116,A -85,B 0,C 180,E1 -8044.505,E2 -8044.505} C_VEL
LIN {X 0,Y 460.5,Z 222.126,A -85,B 0,C 180,E1 -8047.623,E2 -8047.623} C_VEL
LIN {X 0,Y 460.537,Z 222.116,A -85,B 0,C 180,E1 -8050.269,E2 -8050.269} C_VEL
LIN {X 0,Y 460.509,Z 222.125,A -85,B 0,C 180,E1 -8053.374,E2 -8053.374} C_VEL
LIN {X 0,Y 460.509,Z 222.119,A -85,B 0,C 180,E1 -8056.626,E2 -8056.626} C_VEL
LIN {X 0,Y 460.535,Z 222.119,A -85,B 0,C 180,E1 -8059.732,E2 -8059.732} C_VEL
LIN {X 0,Y 460.497,Z 222.118,A -85,B 0,C 180,E1 -8062.524,E2 -8062.524} C_VEL
LIN {X 0,Y 460.537,Z 222.117,A -85,B 0,C 180,E1 -8065.623,E2 -8065.623} C_VEL
LIN {X 0,Y 460.538,Z 222.115,A -85,B 0,C 180,E1 -8068.745,E2 -8068.745} C_VEL
LIN {X 0,Y 460.551,Z 222.113,A -85,B 0,C 180,E1 -8072.261,E2 -8072.261} C_VEL
LIN {X 0,Y 460.541,Z 222.111,A -85,B 0,C 180,E1 -8074.704,E2 -8074.704} C_VEL
LIN {X 0,Y 460.512,Z 222.121,A -85,B 0,C 180,E1 -8077.571,E2 -8077.571} C_VEL
LIN {X 0,Y 460.569,Z 222.11,A -85,B 0,C 180,E1 -8080.384,E2 -8080.384} C_VEL
LIN {X 0,Y 460.605,Z 222.106,A -85,B 0,C 180,E1 -8084.059,E2 -8084.059} C_VEL
LIN {X 0,Y 460.61,Z 222.106,A -85,B 0,C 180,E1 -8087.666,E2 -8087.666} C_VEL
LIN {X 0,Y 460.628,Z 222.108,A -85,B 0,C 180,E1 -8091.224,E2 -8091.224} C_VEL
LIN {X 0,Y 460.709,Z 222.094,A -85,B 0,C 180,E1 -8093.87,E2 -8093.87} C_VEL
LIN {X 0,Y 460.789,Z 222.086,A -85,B 0,C 180,E1 -8097.378,E2 -8097.378} C_VEL
LIN {X 0,Y 460.852,Z 222.076,A -85,B 0,C 180,E1 -8100,E2 -8100} C_VEL
LIN {X 0,Y 460.793,Z 222.08,A -85,B 0,C 180,E1 -8102.623,E2 -8102.623} C_VEL
LIN {X 0,Y 460.688,Z 222.096,A -85,B 0,C 180,E1 -8106.13,E2 -8106.13} C_VEL
LIN {X 0,Y 460.62,Z 222.1,A -85,B 0,C 180,E1 -8108.776,E2 -8108.776} C_VEL
LIN {X 0,Y 460.611,Z 222.103,A -85,B 0,C 180,E1 -8112.334,E2 -8112.334} C_VEL
LIN {X 0,Y 460.602,Z 222.107,A -85,B 0,C 180,E1 -8115.998,E2 -8115.998} C_VEL
LIN {X 0,Y 460.568,Z 222.115,A -85,B 0,C 180,E1 -8119.616,E2 -8119.616} C_VEL
LIN {X 0,Y 460.511,Z 222.113,A -85,B 0,C 180,E1 -8122.429,E2 -8122.429} C_VEL
LIN {X 0,Y 460.547,Z 222.112,A -85,B 0,C 180,E1 -8125.796,E2 -8125.796} C_VEL
LIN {X 0,Y 460.55,Z 222.113,A -85,B 0,C 180,E1 -8128.233,E2 -8128.233} C_VEL
LIN {X 0,Y 460.522,Z 222.121,A -85,B 0,C 180,E1 -8131.283,E2 -8131.283} C_VEL
LIN {X 0,Y 460.532,Z 222.115,A -85,B 0,C 180,E1 -8134.505,E2 -8134.505} C_VEL
LIN {X 0,Y 460.5,Z 222.124,A -85,B 0,C 180,E1 -8137.624,E2 -8137.624} C_VEL
LIN {X 0,Y 460.538,Z 222.115,A -85,B 0,C 180,E1 -8140.269,E2 -8140.269} C_VEL
LIN {X 0,Y 460.51,Z 222.125,A -85,B 0,C 180,E1 -8143.375,E2 -8143.375} C_VEL
LIN {X 0,Y 460.51,Z 222.116,A -85,B 0,C 180,E1 -8146.626,E2 -8146.626} C_VEL
LIN {X 0,Y 460.536,Z 222.118,A -85,B 0,C 180,E1 -8149.732,E2 -8149.732} C_VEL
LIN {X 0,Y 460.501,Z 222.123,A -85,B 0,C 180,E1 -8152.524,E2 -8152.524} C_VEL
LIN {X 0,Y 460.539,Z 222.121,A -85,B 0,C 180,E1 -8155.623,E2 -8155.623} C_VEL
LIN {X 0,Y 460.54,Z 222.116,A -85,B 0,C 180,E1 -8158.745,E2 -8158.745} C_VEL
LIN {X 0,Y 460.568,Z 222.214,A -85,B 0,C 180,E1 -8162.054,E2 -8162.054} C_VEL
LIN {X 0,Y 461.981,Z 230.447,A -85,B 0,C 180,E1 -8163.839,E2 -8163.839} C_VEL
LIN {X 0,Y 461.612,Z 244.385,A -85,B 0,C 180,E1 -8166.657,E2 -8166.657} C_VEL
LIN {X 0,Y 464.846,Z 260.479,A -85,B 0,C 180,E1 -8167.054,E2 -8167.054} C_VEL
LIN {X 0,Y 464.34,Z 315.8,A -85,B 0,C 180,E1 -8167.916,E2 -8167.916} C_VEL
LIN {X 0,Y 463.672,Z 321.651,A -85,B 0,C 180,E1 -8167.981,E2 -8167.981} C_VEL
LIN {X 0,Y 457.954,Z 340.661,A -85,B 0,C 180,E1 -8168.051,E2 -8168.051} C_VEL
LIN {X 0,Y 457.269,Z 346.498,A -85,B 0,C 180,E1 -8168.129,E2 -8168.129} C_VEL
LIN {X 0,Y 457.029,Z 359.36,A -85,B 0,C 180,E1 -8168.431,E2 -8168.431} C_VEL
LIN {X 0,Y 456.65,Z 372.281,A -85,B 0,C 180,E1 -8168.915,E2 -8168.915} C_VEL
LIN {X 0,Y 456.185,Z 383.631,A -85,B 0,C 180,E1 -8169.506,E2 -8169.506} C_VEL
LIN {X 0,Y 455.679,Z 395.279,A -85,B 0,C 180,E1 -8170.307,E2 -8170.307} C_VEL
LIN {X 0,Y 454.986,Z 406.743,A -85,B 0,C 180,E1 -8171.306,E2 -8171.306} C_VEL
LIN {X 0,Y 454.565,Z 415.211,A -85,B 0,C 180,E1 -8172.221,E2 -8172.221} C_VEL
LIN {X 0,Y 454.052,Z 423.984,A -85,B 0,C 180,E1 -8173.361,E2 -8173.361} C_VEL
LIN {X 0,Y 453.53,Z 432.441,A -85,B 0,C 180,E1 -8174.726,E2 -8174.726} C_VEL
LIN {X 0,Y 453.162,Z 439.219,A -85,B 0,C 180,E1 -8176.091,E2 -8176.091} C_VEL
LIN {X 0,Y 452.91,Z 444.607,A -85,B 0,C 180,E1 -8177.453,E2 -8177.453} C_VEL
LIN {X 0,Y 452.679,Z 448.79,A -85,B 0,C 180,E1 -8178.81,E2 -8178.81} C_VEL
LIN {X 0,Y 452.488,Z 451.894,A -85,B 0,C 180,E1 -8180.163,E2 -8180.163} C_VEL
LIN {X 0,Y 452.461,Z 453.432,A -85,B 0,C 180,E1 -8181.064,E2 -8181.064} C_VEL
LIN {X 0,Y 452.464,Z 454.515,A -85,B 0,C 180,E1 -8181.964,E2 -8181.964} C_VEL
LIN {X 0,Y 452.517,Z 455.486,A -85,B 0,C 180,E1 -8183.759,E2 -8183.759} C_VEL
LIN {X 0,Y 452.476,Z 455.397,A -85,B 0,C 180,E1 -8184.653,E2 -8184.653} C_VEL
LIN {X 0,Y 452.475,Z 453.963,A -85,B 0,C 180,E1 -8186.438,E2 -8186.438} C_VEL
LIN {X 0,Y 452.543,Z 452.658,A -85,B 0,C 180,E1 -8187.33,E2 -8187.33} C_VEL
LIN {X 0,Y 452.574,Z 449.904,A -85,B 0,C 180,E1 -8188.665,E2 -8188.665} C_VEL
LIN {X 0,Y 452.616,Z 446.146,A -85,B 0,C 180,E1 -8190,E2 -8190} C_VEL
LIN {X 0,Y 452.88,Z 441.27,A -85,B 0,C 180,E1 -8191.334,E2 -8191.334} C_VEL
LIN {X 0,Y 453.116,Z 435.151,A -85,B 0,C 180,E1 -8192.667,E2 -8192.667} C_VEL
LIN {X 0,Y 453.419,Z 428.904,A -85,B 0,C 180,E1 -8193.777,E2 -8193.777} C_VEL
LIN {X 0,Y 453.915,Z 421.403,A -85,B 0,C 180,E1 -8194.885,E2 -8194.885} C_VEL
LIN {X 0,Y 454.475,Z 412.333,A -85,B 0,C 180,E1 -8195.992,E2 -8195.992} C_VEL
LIN {X 0,Y 455.013,Z 402.271,A -85,B 0,C 180,E1 -8196.986,E2 -8196.986} C_VEL
LIN {X 0,Y 455.547,Z 391.12,A -85,B 0,C 180,E1 -8197.87,E2 -8197.87} C_VEL
LIN {X 0,Y 455.948,Z 380.584,A -85,B 0,C 180,E1 -8198.532,E2 -8198.532} C_VEL
LIN {X 0,Y 456.401,Z 367.867,A -85,B 0,C 180,E1 -8199.137,E2 -8199.137} C_VEL
LIN {X 0,Y 456.646,Z 355.114,A -85,B 0,C 180,E1 -8199.551,E2 -8199.551} C_VEL
LIN {X 0,Y 456.915,Z 336.411,A -85,B 0,C 180,E1 -8199.891,E2 -8199.891} C_VEL
LIN {X 0,Y 457.425,Z 260.342,A -85,B 0,C 180,E1 -8201.088,E2 -8201.088} C_VEL
LIN {X 0,Y 454.498,Z 244.486,A -85,B 0,C 180,E1 -8201.455,E2 -8201.455} C_VEL
LIN {X 0,Y 454.844,Z 230.419,A -85,B 0,C 180,E1 -8204.313,E2 -8204.313} C_VEL
LIN {X 0,Y 453.582,Z 222.987,A -85,B 0,C 180,E1 -8205.945,E2 -8205.945} C_VEL
LIN {X 0,Y 453.521,Z 222.994,A -85,B 0,C 180,E1 -8209.039,E2 -8209.039} C_VEL
LIN {X 0,Y 453.48,Z 222.993,A -85,B 0,C 180,E1 -8211.836,E2 -8211.836} C_VEL
LIN {X 0,Y 453.504,Z 222.998,A -85,B 0,C 180,E1 -8214.735,E2 -8214.735} C_VEL
LIN {X 0,Y 453.509,Z 222.99,A -85,B 0,C 180,E1 -8217.953,E2 -8217.953} C_VEL
LIN {X 0,Y 453.478,Z 223,A -85,B 0,C 180,E1 -8220.759,E2 -8220.759} C_VEL
LIN {X 0,Y 453.479,Z 222.993,A -85,B 0,C 180,E1 -8223.912,E2 -8223.912} C_VEL
LIN {X 0,Y 453.454,Z 222.998,A -85,B 0,C 180,E1 -8227.19,E2 -8227.19} C_VEL
LIN {X 0,Y 453.488,Z 222.992,A -85,B 0,C 180,E1 -8229.45,E2 -8229.45} C_VEL
LIN {X 0,Y 453.478,Z 222.994,A -85,B 0,C 180,E1 -8231.935,E2 -8231.935} C_VEL
LIN {X 0,Y 453.484,Z 222.993,A -85,B 0,C 180,E1 -8235.471,E2 -8235.471} C_VEL
LIN {X 0,Y 453.465,Z 222.997,A -85,B 0,C 180,E1 -8238.207,E2 -8238.207} C_VEL
LIN {X 0,Y 453.491,Z 222.998,A -85,B 0,C 180,E1 -8240.794,E2 -8240.794} C_VEL
LIN {X 0,Y 453.452,Z 222.997,A -85,B 0,C 180,E1 -8243.917,E2 -8243.917} C_VEL
LIN {X 0,Y 453.484,Z 222.994,A -85,B 0,C 180,E1 -8247.151,E2 -8247.151} C_VEL
LIN {X 0,Y 453.475,Z 222.997,A -85,B 0,C 180,E1 -8250.268,E2 -8250.268} C_VEL
LIN {X 0,Y 453.533,Z 222.99,A -85,B 0,C 180,E1 -8252.297,E2 -8252.297} C_VEL
LIN {X 0,Y 453.493,Z 222.992,A -85,B 0,C 180,E1 -8255.264,E2 -8255.264} C_VEL
LIN {X 0,Y 453.481,Z 222.998,A -85,B 0,C 180,E1 -8258.415,E2 -8258.415} C_VEL
LIN {X 0,Y 453.523,Z 222.991,A -85,B 0,C 180,E1 -8261.008,E2 -8261.008} C_VEL
LIN {X 0,Y 453.57,Z 222.982,A -85,B 0,C 180,E1 -8263.88,E2 -8263.88} C_VEL
LIN {X 0,Y 453.565,Z 222.982,A -85,B 0,C 180,E1 -8267.471,E2 -8267.471} C_VEL
LIN {X 0,Y 453.585,Z 222.982,A -85,B 0,C 180,E1 -8271.086,E2 -8271.086} C_VEL
LIN {X 0,Y 453.653,Z 222.971,A -85,B 0,C 180,E1 -8273.774,E2 -8273.774} C_VEL
LIN {X 0,Y 453.744,Z 222.961,A -85,B 0,C 180,E1 -8277.337,E2 -8277.337} C_VEL
LIN {X 0,Y 453.822,Z 222.951,A -85,B 0,C 180,E1 -8280,E2 -8280} C_VEL
LIN {X 0,Y 453.737,Z 222.968,A -85,B 0,C 180,E1 -8282.663,E2 -8282.663} C_VEL
LIN {X 0,Y 453.677,Z 222.972,A -85,B 0,C 180,E1 -8286.225,E2 -8286.225} C_VEL
LIN {X 0,Y 453.591,Z 222.983,A -85,B 0,C 180,E1 -8288.913,E2 -8288.913} C_VEL
LIN {X 0,Y 453.564,Z 222.99,A -85,B 0,C 180,E1 -8292.529,E2 -8292.529} C_VEL
LIN {X 0,Y 453.545,Z 222.988,A -85,B 0,C 180,E1 -8296.196,E2 -8296.196} C_VEL
LIN {X 0,Y 453.518,Z 222.991,A -85,B 0,C 180,E1 -8299.039,E2 -8299.039} C_VEL
LIN {X 0,Y 453.477,Z 222.994,A -85,B 0,C 180,E1 -8301.836,E2 -8301.836} C_VEL
LIN {X 0,Y 453.502,Z 222.996,A -85,B 0,C 180,E1 -8304.735,E2 -8304.735} C_VEL
LIN {X 0,Y 453.506,Z 222.991,A -85,B 0,C 180,E1 -8307.953,E2 -8307.953} C_VEL
LIN {X 0,Y 453.476,Z 222.999,A -85,B 0,C 180,E1 -8310.76,E2 -8310.76} C_VEL
LIN {X 0,Y 453.468,Z 222.995,A -85,B 0,C 180,E1 -8313.914,E2 -8313.914} C_VEL
LIN {X 0,Y 453.45,Z 222.998,A -85,B 0,C 180,E1 -8317.19,E2 -8317.19} C_VEL
LIN {X 0,Y 453.494,Z 222.999,A -85,B 0,C 180,E1 -8320.609,E2 -8320.609} C_VEL
LIN {X 0,Y 453.46,Z 222.999,A -85,B 0,C 180,E1 -8324.222,E2 -8324.222} C_VEL
LIN {X 0,Y 453.449,Z 222.999,A -85,B 0,C 180,E1 -8327.003,E2 -8327.003} C_VEL
LIN {X 0,Y 453.494,Z 222.991,A -85,B 0,C 180,E1 -8329.409,E2 -8329.409} C_VEL
LIN {X 0,Y 453.447,Z 223.001,A -85,B 0,C 180,E1 -8332.228,E2 -8332.228} C_VEL
LIN {X 0,Y 453.488,Z 222.993,A -85,B 0,C 180,E1 -8335.223,E2 -8335.223} C_VEL
LIN {X 0,Y 453.467,Z 223.002,A -85,B 0,C 180,E1 -8338.475,E2 -8338.475} C_VEL
LIN {X 0,Y 453.53,Z 222.992,A -85,B 0,C 180,E1 -8342.041,E2 -8342.041} C_VEL
LIN {X 0,Y 453.512,Z 223.018,A -85,B 0,C 180,E1 -8344.191,E2 -8344.191} C_VEL
LIN {X 0,Y 455.709,Z 235.259,A -85,B 0,C 180,E1 -8346.602,E2 -8346.602} C_VEL
LIN {X 0,Y 455.008,Z 250.672,A -85,B 0,C 180,E1 -8349.427,E2 -8349.427} C_VEL
LIN {X 0,Y 454.274,Z 267.991,A -85,B 0,C 180,E1 -8352.566,E2 -8352.566} C_VEL
LIN {X 0,Y 457.35,Z 289.457,A -85,B 0,C 180,E1 -8353.024,E2 -8353.024} C_VEL
LIN {X 0,Y 456.686,Z 376.234,A -85,B 0,C 180,E1 -8354.405,E2 -8354.405} C_VEL
LIN {X 0,Y 456.29,Z 388.769,A -85,B 0,C 180,E1 -8354.763,E2 -8354.763} C_VEL
LIN {X 0,Y 455.759,Z 401.724,A -85,B 0,C 180,E1 -8355.317,E2 -8355.317} C_VEL
LIN {X 0,Y 455.233,Z 414.02,A -85,B 0,C 180,E1 -8356.041,E2 -8356.041} C_VEL
LIN {X 0,Y 454.588,Z 426.233,A -85,B 0,C 180,E1 -8356.984,E2 -8356.984} C_VEL
LIN {X 0,Y 454.215,Z 436.108,A -85,B 0,C 180,E1 -8357.943,E2 -8357.943} C_VEL
LIN {X 0,Y 453.663,Z 445.502,A -85,B 0,C 180,E1 -8359.06,E2 -8359.06} C_VEL
LIN {X 0,Y 453.201,Z 454.582,A -85,B 0,C 180,E1 -8360.404,E2 -8360.404} C_VEL
LIN {X 0,Y 452.906,Z 461.897,A -85,B 0,C 180,E1 -8361.747,E2 -8361.747} C_VEL
LIN {X 0,Y 452.692,Z 466.841,A -85,B 0,C 180,E1 -8362.866,E2 -8362.866} C_VEL
LIN {X 0,Y 452.557,Z 471.641,A -85,B 0,C 180,E1 -8364.207,E2 -8364.207} C_VEL
LIN {X 0,Y 452.485,Z 475.316,A -85,B 0,C 180,E1 -8365.546,E2 -8365.546} C_VEL
LIN {X 0,Y 452.48,Z 477.215,A -85,B 0,C 180,E1 -8366.438,E2 -8366.438} C_VEL
LIN {X 0,Y 452.508,Z 478.658,A -85,B 0,C 180,E1 -8367.329,E2 -8367.329} C_VEL
LIN {X 0,Y 452.428,Z 480.308,A -85,B 0,C 180,E1 -8369.11,E2 -8369.11} C_VEL
LIN {X 0,Y 452.436,Z 480.554,A -85,B 0,C 180,E1 -8370,E2 -8370} C_VEL
LIN {X 0,Y 452.428,Z 480.379,A -85,B 0,C 180,E1 -8370.89,E2 -8370.89} C_VEL
LIN {X 0,Y 452.508,Z 478.825,A -85,B 0,C 180,E1 -8372.671,E2 -8372.671} C_VEL
LIN {X 0,Y 452.479,Z 477.459,A -85,B 0,C 180,E1 -8373.562,E2 -8373.562} C_VEL
LIN {X 0,Y 452.544,Z 474.576,A -85,B 0,C 180,E1 -8374.9,E2 -8374.9} C_VEL
LIN {X 0,Y 452.61,Z 470.159,A -85,B 0,C 180,E1 -8376.396,E2 -8376.396} C_VEL
LIN {X 0,Y 452.802,Z 465.635,A -85,B 0,C 180,E1 -8377.581,E2 -8377.581} C_VEL
LIN {X 0,Y 453.092,Z 459.323,A -85,B 0,C 180,E1 -8378.923,E2 -8378.923} C_VEL
LIN {X 0,Y 453.474,Z 451.426,A -85,B 0,C 180,E1 -8380.267,E2 -8380.267} C_VEL
LIN {X 0,Y 453.995,Z 443.395,A -85,B 0,C 180,E1 -8381.384,E2 -8381.384} C_VEL
LIN {X 0,Y 454.566,Z 433.611,A -85,B 0,C 180,E1 -8382.501,E2 -8382.501} C_VEL
LIN {X 0,Y 455.098,Z 422.715,A -85,B 0,C 180,E1 -8383.508,E2 -8383.508} C_VEL
LIN {X 0,Y 455.758,Z 410.288,A -85,B 0,C 180,E1 -8384.398,E2 -8384.398} C_VEL
LIN {X 0,Y 456.356,Z 398.097,A -85,B 0,C 180,E1 -8385.063,E2 -8385.063} C_VEL
LIN {X 0,Y 456.874,Z 385.315,A -85,B 0,C 180,E1 -8385.559,E2 -8385.559} C_VEL
LIN {X 0,Y 457.183,Z 371.808,A -85,B 0,C 180,E1 -8385.892,E2 -8385.892} C_VEL
LIN {X 0,Y 457.792,Z 287.465,A -85,B 0,C 180,E1 -8387.237,E2 -8387.237} C_VEL
LIN {X 0,Y 454.494,Z 267.903,A -85,B 0,C 180,E1 -8387.701,E2 -8387.701} C_VEL
LIN {X 0,Y 455.301,Z 251.071,A -85,B 0,C 180,E1 -8390.795,E2 -8390.795} C_VEL
LIN {X 0,Y 456.038,Z 237.204,A -85,B 0,C 180,E1 -8393.38,E2 -8393.38} C_VEL
LIN {X 0,Y 455.138,Z 230.897,A -85,B 0,C 180,E1 -8394.64,E2 -8394.64} C_VEL
LIN {X 0,Y 453.487,Z 223,A -85,B 0,C 180,E1 -8396.309,E2 -8396.309} C_VEL
LIN {X 0,Y 453.494,Z 222.998,A -85,B 0,C 180,E1 -8398.713,E2 -8398.713} C_VEL
LIN {X 0,Y 453.466,Z 223.001,A -85,B 0,C 180,E1 -8401.799,E2 -8401.799} C_VEL
LIN {X 0,Y 453.48,Z 222.997,A -85,B 0,C 180,E1 -8404.989,E2 -8404.989} C_VEL
LIN {X 0,Y 453.46,Z 222.997,A -85,B 0,C 180,E1 -8408.312,E2 -8408.312} C_VEL
LIN {X 0,Y 453.494,Z 222.993,A -85,B 0,C 180,E1 -8410.609,E2 -8410.609} C_VEL
LIN {X 0,Y 453.461,Z 222.997,A -85,B 0,C 180,E1 -8414.222,E2 -8414.222} C_VEL
LIN {X 0,Y 453.449,Z 223.001,A -85,B 0,C 180,E1 -8417.003,E2 -8417.003} C_VEL
LIN {X 0,Y 453.494,Z 222.998,A -85,B 0,C 180,E1 -8419.409,E2 -8419.409} C_VEL
LIN {X 0,Y 453.45,Z 222.997,A -85,B 0,C 180,E1 -8422.81,E2 -8422.81} C_VEL
LIN {X 0,Y 453.468,Z 222.993,A -85,B 0,C 180,E1 -8426.087,E2 -8426.087} C_VEL
LIN {X 0,Y 453.476,Z 222.999,A -85,B 0,C 180,E1 -8429.24,E2 -8429.24} C_VEL
LIN {X 0,Y 453.508,Z 222.99,A -85,B 0,C 180,E1 -8432.296,E2 -8432.296} C_VEL
LIN {X 0,Y 453.501,Z 222.992,A -85,B 0,C 180,E1 -8435.265,E2 -8435.265} C_VEL
LIN {X 0,Y 453.481,Z 222.99,A -85,B 0,C 180,E1 -8438.415,E2 -8438.415} C_VEL
LIN {X 0,Y 453.523,Z 222.991,A -85,B 0,C 180,E1 -8441.009,E2 -8441.009} C_VEL
LIN {X 0,Y 453.57,Z 222.983,A -85,B 0,C 180,E1 -8443.88,E2 -8443.88} C_VEL
LIN {X 0,Y 453.565,Z 222.985,A -85,B 0,C 180,E1 -8447.471,E2 -8447.471} C_VEL
LIN {X 0,Y 453.591,Z 222.983,A -85,B 0,C 180,E1 -8451.087,E2 -8451.087} C_VEL
LIN {X 0,Y 453.677,Z 222.971,A -85,B 0,C 180,E1 -8453.775,E2 -8453.775} C_VEL
LIN {X 0,Y 453.733,Z 222.965,A -85,B 0,C 180,E1 -8457.337,E2 -8457.337} C_VEL
LIN {X 0,Y 453.822,Z 222.952,A -85,B 0,C 180,E1 -8460,E2 -8460} C_VEL
LIN {X 0,Y 453.737,Z 222.959,A -85,B 0,C 180,E1 -8462.663,E2 -8462.663} C_VEL
LIN {X 0,Y 453.653,Z 222.972,A -85,B 0,C 180,E1 -8466.226,E2 -8466.226} C_VEL
LIN {X 0,Y 453.586,Z 222.977,A -85,B 0,C 180,E1 -8468.914,E2 -8468.914} C_VEL
LIN {X 0,Y 453.565,Z 222.981,A -85,B 0,C 180,E1 -8472.529,E2 -8472.529} C_VEL
LIN {X 0,Y 453.546,Z 222.985,A -85,B 0,C 180,E1 -8476.196,E2 -8476.196} C_VEL
LIN {X 0,Y 453.518,Z 222.987,A -85,B 0,C 180,E1 -8479.039,E2 -8479.039} C_VEL
LIN {X 0,Y 453.478,Z 222.991,A -85,B 0,C 180,E1 -8481.836,E2 -8481.836} C_VEL
LIN {X 0,Y 453.493,Z 222.992,A -85,B 0,C 180,E1 -8484.736,E2 -8484.736} C_VEL
LIN {X 0,Y 453.53,Z 222.989,A -85,B 0,C 180,E1 -8487.959,E2 -8487.959} C_VEL
LIN {X 0,Y 453.467,Z 223.002,A -85,B 0,C 180,E1 -8491.525,E2 -8491.525} C_VEL
LIN {X 0,Y 453.488,Z 222.994,A -85,B 0,C 180,E1 -8494.777,E2 -8494.777} C_VEL
LIN {X 0,Y 453.46,Z 222.996,A -85,B 0,C 180,E1 -8498.312,E2 -8498.312} C_VEL
LIN {X 0,Y 453.495,Z 222.993,A -85,B 0,C 180,E1 -8500.609,E2 -8500.609} C_VEL
LIN {X 0,Y 453.462,Z 222.997,A -85,B 0,C 180,E1 -8504.222,E2 -8504.222} C_VEL
LIN {X 0,Y 453.45,Z 222.998,A -85,B 0,C 180,E1 -8507.003,E2 -8507.003} C_VEL
LIN {X 0,Y 453.495,Z 222.998,A -85,B 0,C 180,E1 -8509.409,E2 -8509.409} C_VEL
LIN {X 0,Y 453.454,Z 223.002,A -85,B 0,C 180,E1 -8512.81,E2 -8512.81} C_VEL
LIN {X 0,Y 453.471,Z 222.998,A -85,B 0,C 180,E1 -8516.087,E2 -8516.087} C_VEL
LIN {X 0,Y 453.478,Z 222.997,A -85,B 0,C 180,E1 -8519.241,E2 -8519.241} C_VEL
LIN {X 0,Y 453.511,Z 223.057,A -85,B 0,C 180,E1 -8521.813,E2 -8521.813} C_VEL
LIN {X 0,Y 455.009,Z 231.235,A -85,B 0,C 180,E1 -8523.62,E2 -8523.62} C_VEL
LIN {X 0,Y 454.797,Z 242.803,A -85,B 0,C 180,E1 -8526,E2 -8526} C_VEL
LIN {X 0,Y 454.727,Z 244.548,A -85,B 0,C 180,E1 -8526.354,E2 -8526.354} C_VEL
LIN {X 0,Y 458.085,Z 261.207,A -85,B 0,C 180,E1 -8526.778,E2 -8526.778} C_VEL
LIN {X 0,Y 457.269,Z 346.498,A -85,B 0,C 180,E1 -8528.129,E2 -8528.129} C_VEL
LIN {X 0,Y 456.888,Z 350.396,A -85,B 0,C 180,E1 -8528.189,E2 -8528.189} C_VEL
LIN {X 0,Y 454.845,Z 358.007,A -85,B 0,C 180,E1 -8528.301,E2 -8528.301} C_VEL
LIN {X 0,Y 450.957,Z 369.098,A -85,B 0,C 180,E1 -8528.547,E2 -8528.547} C_VEL
LIN {X 0,Y 449.839,Z 374.671,A -85,B 0,C 180,E1 -8528.761,E2 -8528.761} C_VEL
LIN {X 0,Y 449.72,Z 376.471,A -85,B 0,C 180,E1 -8528.85,E2 -8528.85} C_VEL
LIN {X 0,Y 449.22,Z 387.774,A -85,B 0,C 180,E1 -8529.509,E2 -8529.509} C_VEL
LIN {X 0,Y 448.6,Z 399.426,A -85,B 0,C 180,E1 -8530.388,E2 -8530.388} C_VEL
LIN {X 0,Y 447.953,Z 409.614,A -85,B 0,C 180,E1 -8531.357,E2 -8531.357} C_VEL
LIN {X 0,Y 447.418,Z 418.553,A -85,B 0,C 180,E1 -8532.4,E2 -8532.4} C_VEL
LIN {X 0,Y 446.819,Z 428.062,A -85,B 0,C 180,E1 -8533.762,E2 -8533.762} C_VEL
LIN {X 0,Y 446.353,Z 435.864,A -85,B 0,C 180,E1 -8535.175,E2 -8535.175} C_VEL
LIN {X 0,Y 445.964,Z 442.895,A -85,B 0,C 180,E1 -8536.791,E2 -8536.791} C_VEL
LIN {X 0,Y 445.73,Z 447.526,A -85,B 0,C 180,E1 -8538.172,E2 -8538.172} C_VEL
LIN {X 0,Y 445.581,Z 449.965,A -85,B 0,C 180,E1 -8539.09,E2 -8539.09} C_VEL
LIN {X 0,Y 445.423,Z 451.95,A -85,B 0,C 180,E1 -8540.005,E2 -8540.005} C_VEL
LIN {X 0,Y 445.391,Z 453.516,A -85,B 0,C 180,E1 -8540.921,E2 -8540.921} C_VEL
LIN {X 0,Y 445.364,Z 454.649,A -85,B 0,C 180,E1 -8541.835,E2 -8541.835} C_VEL
LIN {X 0,Y 445.415,Z 455.67,A -85,B 0,C 180,E1 -8543.659,E2 -8543.659} C_VEL
LIN {X 0,Y 445.396,Z 455.608,A -85,B 0,C 180,E1 -8544.567,E2 -8544.567} C_VEL
LIN {X 0,Y 445.36,Z 455.139,A -85,B 0,C 180,E1 -8545.474,E2 -8545.474} C_VEL
LIN {X 0,Y 445.464,Z 452.968,A -85,B 0,C 180,E1 -8547.287,E2 -8547.287} C_VEL
LIN {X 0,Y 445.501,Z 450.266,A -85,B 0,C 180,E1 -8548.644,E2 -8548.644} C_VEL
LIN {X 0,Y 445.543,Z 446.565,A -85,B 0,C 180,E1 -8550,E2 -8550} C_VEL
LIN {X 0,Y 445.793,Z 441.75,A -85,B 0,C 180,E1 -8551.355,E2 -8551.355} C_VEL
LIN {X 0,Y 446.051,Z 435.695,A -85,B 0,C 180,E1 -8552.709,E2 -8552.709} C_VEL
LIN {X 0,Y 446.365,Z 429.521,A -85,B 0,C 180,E1 -8553.837,E2 -8553.837} C_VEL
LIN {X 0,Y 447.002,Z 420.477,A -85,B 0,C 180,E1 -8555.187,E2 -8555.187} C_VEL
LIN {X 0,Y 447.603,Z 410.04,A -85,B 0,C 180,E1 -8556.423,E2 -8556.423} C_VEL
LIN {X 0,Y 448.223,Z 399.421,A -85,B 0,C 180,E1 -8557.432,E2 -8557.432} C_VEL
LIN {X 0,Y 448.696,Z 389.153,A -85,B 0,C 180,E1 -8558.217,E2 -8558.217} C_VEL
LIN {X 0,Y 449.202,Z 376.858,A -85,B 0,C 180,E1 -8558.944,E2 -8558.944} C_VEL
LIN {X 0,Y 449.61,Z 363.919,A -85,B 0,C 180,E1 -8559.503,E2 -8559.503} C_VEL
LIN {X 0,Y 449.872,Z 351.239,A -85,B 0,C 180,E1 -8559.867,E2 -8559.867} C_VEL
LIN {X 0,Y 450.635,Z 261.406,A -85,B 0,C 180,E1 -8561.312,E2 -8561.312} C_VEL
LIN {X 0,Y 447.526,Z 244.592,A -85,B 0,C 180,E1 -8561.723,E2 -8561.723} C_VEL
LIN {X 0,Y 447.889,Z 232.012,A -85,B 0,C 180,E1 -8564.308,E2 -8564.308} C_VEL
LIN {X 0,Y 446.526,Z 223.867,A -85,B 0,C 180,E1 -8566.104,E2 -8566.104} C_VEL
LIN {X 0,Y 446.472,Z 223.869,A -85,B 0,C 180,E1 -8569.303,E2 -8569.303} C_VEL
LIN {X 0,Y 446.421,Z 223.874,A -85,B 0,C 180,E1 -8572.199,E2 -8572.199} C_VEL
LIN {X 0,Y 446.446,Z 223.871,A -85,B 0,C 180,E1 -8575.153,E2 -8575.153} C_VEL
LIN {X 0,Y 446.452,Z 223.87,A -85,B 0,C 180,E1 -8578.181,E2 -8578.181} C_VEL
LIN {X 0,Y 446.418,Z 223.874,A -85,B 0,C 180,E1 -8581.3,E2 -8581.3} C_VEL
LIN {X 0,Y 446.431,Z 223.877,A -85,B 0,C 180,E1 -8584.523,E2 -8584.523} C_VEL
LIN {X 0,Y 446.416,Z 223.874,A -85,B 0,C 180,E1 -8588.079,E2 -8588.079} C_VEL
LIN {X 0,Y 446.429,Z 223.876,A -85,B 0,C 180,E1 -8590.917,E2 -8590.917} C_VEL
LIN {X 0,Y 446.401,Z 223.875,A -85,B 0,C 180,E1 -8593.846,E2 -8593.846} C_VEL
LIN {X 0,Y 446.399,Z 223.879,A -85,B 0,C 180,E1 -8596.403,E2 -8596.403} C_VEL
LIN {X 0,Y 446.443,Z 223.87,A -85,B 0,C 180,E1 -8599.802,E2 -8599.802} C_VEL
LIN {X 0,Y 446.401,Z 223.876,A -85,B 0,C 180,E1 -8603.254,E2 -8603.254} C_VEL
LIN {X 0,Y 446.449,Z 223.876,A -85,B 0,C 180,E1 -8606.566,E2 -8606.566} C_VEL
LIN {X 0,Y 446.432,Z 223.872,A -85,B 0,C 180,E1 -8609.979,E2 -8609.979} C_VEL
LIN {X 0,Y 446.464,Z 223.872,A -85,B 0,C 180,E1 -8612.838,E2 -8612.838} C_VEL
LIN {X 0,Y 446.461,Z 223.868,A -85,B 0,C 180,E1 -8615.925,E2 -8615.925} C_VEL
LIN {X 0,Y 446.454,Z 223.874,A -85,B 0,C 180,E1 -8618.773,E2 -8618.773} C_VEL
LIN {X 0,Y 446.451,Z 223.868,A -85,B 0,C 180,E1 -8621.649,E2 -8621.649} C_VEL
LIN {X 0,Y 446.507,Z 223.868,A -85,B 0,C 180,E1 -8624.48,E2 -8624.48} C_VEL
LIN {X 0,Y 446.518,Z 223.863,A -85,B 0,C 180,E1 -8628.193,E2 -8628.193} C_VEL
LIN {X 0,Y 446.533,Z 223.862,A -85,B 0,C 180,E1 -8630.944,E2 -8630.944} C_VEL
LIN {X 0,Y 446.621,Z 223.847,A -85,B 0,C 180,E1 -8633.676,E2 -8633.676} C_VEL
LIN {X 0,Y 446.691,Z 223.839,A -85,B 0,C 180,E1 -8637.295,E2 -8637.295} C_VEL
LIN {X 0,Y 446.792,Z 223.827,A -85,B 0,C 180,E1 -8640,E2 -8640} C_VEL
LIN {X 0,Y 446.683,Z 223.846,A -85,B 0,C 180,E1 -8642.705,E2 -8642.705} C_VEL
LIN {X 0,Y 446.646,Z 223.848,A -85,B 0,C 180,E1 -8646.324,E2 -8646.324} C_VEL
LIN {X 0,Y 446.537,Z 223.86,A -85,B 0,C 180,E1 -8649.055,E2 -8649.055} C_VEL
LIN {X 0,Y 446.522,Z 223.866,A -85,B 0,C 180,E1 -8652.73,E2 -8652.73} C_VEL
LIN {X 0,Y 446.496,Z 223.866,A -85,B 0,C 180,E1 -8656.227,E2 -8656.227} C_VEL
LIN {X 0,Y 446.469,Z 223.867,A -85,B 0,C 180,E1 -8659.303,E2 -8659.303} C_VEL
LIN {X 0,Y 446.419,Z 223.876,A -85,B 0,C 180,E1 -8662.2,E2 -8662.2} C_VEL
LIN {X 0,Y 446.443,Z 223.871,A -85,B 0,C 180,E1 -8665.153,E2 -8665.153} C_VEL
LIN {X 0,Y 446.449,Z 223.872,A -85,B 0,C 180,E1 -8668.181,E2 -8668.181} C_VEL
LIN {X 0,Y 446.416,Z 223.873,A -85,B 0,C 180,E1 -8671.3,E2 -8671.3} C_VEL
LIN {X 0,Y 446.423,Z 223.88,A -85,B 0,C 180,E1 -8674.524,E2 -8674.524} C_VEL
LIN {X 0,Y 446.411,Z 223.876,A -85,B 0,C 180,E1 -8678.079,E2 -8678.079} C_VEL
LIN {X 0,Y 446.419,Z 223.873,A -85,B 0,C 180,E1 -8681.392,E2 -8681.392} C_VEL
LIN {X 0,Y 446.45,Z 223.87,A -85,B 0,C 180,E1 -8685.104,E2 -8685.104} C_VEL
LIN {X 0,Y 446.419,Z 223.88,A -85,B 0,C 180,E1 -8688.608,E2 -8688.608} C_VEL
LIN {X 0,Y 446.437,Z 223.873,A -85,B 0,C 180,E1 -8690.972,E2 -8690.972} C_VEL
LIN {X 0,Y 446.418,Z 223.878,A -85,B 0,C 180,E1 -8694.374,E2 -8694.374} C_VEL
LIN {X 0,Y 446.423,Z 223.872,A -85,B 0,C 180,E1 -8697.639,E2 -8697.639} C_VEL
LIN {X 0,Y 446.448,Z 223.874,A -85,B 0,C 180,E1 -8700.791,E2 -8700.791} C_VEL
LIN {X 0,Y 446.477,Z 223.935,A -85,B 0,C 180,E1 -8704.005,E2 -8704.005} C_VEL
LIN {X 0,Y 448.725,Z 236.181,A -85,B 0,C 180,E1 -8706.46,E2 -8706.46} C_VEL
LIN {X 0,Y 448.103,Z 250.318,A -85,B 0,C 180,E1 -8709.096,E2 -8709.096} C_VEL
LIN {X 0,Y 447.283,Z 267.788,A -85,B 0,C 180,E1 -8712.311,E2 -8712.311} C_VEL
LIN {X 0,Y 450.46,Z 288.997,A -85,B 0,C 180,E1 -8712.779,E2 -8712.779} C_VEL
LIN {X 0,Y 449.804,Z 376.174,A -85,B 0,C 180,E1 -8714.19,E2 -8714.19} C_VEL
LIN {X 0,Y 449.358,Z 389.431,A -85,B 0,C 180,E1 -8714.581,E2 -8714.581} C_VEL
LIN {X 0,Y 448.817,Z 402.168,A -85,B 0,C 180,E1 -8715.143,E2 -8715.143} C_VEL
LIN {X 0,Y 448.333,Z 413.48,A -85,B 0,C 180,E1 -8715.822,E2 -8715.822} C_VEL
LIN {X 0,Y 447.662,Z 425.381,A -85,B 0,C 180,E1 -8716.746,E2 -8716.746} C_VEL
LIN {X 0,Y 447.204,Z 435.682,A -85,B 0,C 180,E1 -8717.751,E2 -8717.751} C_VEL
LIN {X 0,Y 446.672,Z 445.134,A -85,B 0,C 180,E1 -8718.887,E2 -8718.887} C_VEL
LIN {X 0,Y 446.179,Z 454.245,A -85,B 0,C 180,E1 -8720.251,E2 -8720.251} C_VEL
LIN {X 0,Y 445.844,Z 461.586,A -85,B 0,C 180,E1 -8721.616,E2 -8721.616} C_VEL
LIN {X 0,Y 445.618,Z 466.552,A -85,B 0,C 180,E1 -8722.752,E2 -8722.752} C_VEL
LIN {X 0,Y 445.482,Z 470.822,A -85,B 0,C 180,E1 -8723.94,E2 -8723.94} C_VEL
LIN {X 0,Y 445.411,Z 475.067,A -85,B 0,C 180,E1 -8725.475,E2 -8725.475} C_VEL
LIN {X 0,Y 445.379,Z 476.974,A -85,B 0,C 180,E1 -8726.381,E2 -8726.381} C_VEL
LIN {X 0,Y 445.432,Z 478.435,A -85,B 0,C 180,E1 -8727.287,E2 -8727.287} C_VEL
LIN {X 0,Y 445.339,Z 480.1,A -85,B 0,C 180,E1 -8729.096,E2 -8729.096} C_VEL
LIN {X 0,Y 445.343,Z 480.354,A -85,B 0,C 180,E1 -8730,E2 -8730} C_VEL
LIN {X 0,Y 445.339,Z 480.194,A -85,B 0,C 180,E1 -8730.904,E2 -8730.904} C_VEL
LIN {X 0,Y 445.432,Z 478.656,A -85,B 0,C 180,E1 -8732.713,E2 -8732.713} C_VEL
LIN {X 0,Y 445.377,Z 477.298,A -85,B 0,C 180,E1 -8733.619,E2 -8733.619} C_VEL
LIN {X 0,Y 445.473,Z 474.432,A -85,B 0,C 180,E1 -8734.978,E2 -8734.978} C_VEL
LIN {X 0,Y 445.529,Z 470.397,A -85,B 0,C 180,E1 -8736.386,E2 -8736.386} C_VEL
LIN {X 0,Y 445.73,Z 465.53,A -85,B 0,C 180,E1 -8737.702,E2 -8737.702} C_VEL
LIN {X 0,Y 446.023,Z 459.245,A -85,B 0,C 180,E1 -8739.066,E2 -8739.066} C_VEL
LIN {X 0,Y 446.465,Z 451.385,A -85,B 0,C 180,E1 -8740.43,E2 -8740.43} C_VEL
LIN {X 0,Y 447.037,Z 443.388,A -85,B 0,C 180,E1 -8741.563,E2 -8741.563} C_VEL
LIN {X 0,Y 447.635,Z 433.645,A -85,B 0,C 180,E1 -8742.698,E2 -8742.698} C_VEL
LIN {X 0,Y 448.199,Z 422.818,A -85,B 0,C 180,E1 -8743.719,E2 -8743.719} C_VEL
LIN {X 0,Y 448.833,Z 412.244,A -85,B 0,C 180,E1 -8744.509,E2 -8744.509} C_VEL
LIN {X 0,Y 449.45,Z 400.655,A -85,B 0,C 180,E1 -8745.184,E2 -8745.184} C_VEL
LIN {X 0,Y 449.978,Z 387.55,A -85,B 0,C 180,E1 -8745.746,E2 -8745.746} C_VEL
LIN {X 0,Y 450.376,Z 374.457,A -85,B 0,C 180,E1 -8746.109,E2 -8746.109} C_VEL
LIN {X 0,Y 451.09,Z 288.447,A -85,B 0,C 180,E1 -8747.509,E2 -8747.509} C_VEL
LIN {X 0,Y 447.563,Z 267.652,A -85,B 0,C 180,E1 -8748.022,E2 -8748.022} C_VEL
LIN {X 0,Y 448.491,Z 249.77,A -85,B 0,C 180,E1 -8751.367,E2 -8751.367} C_VEL
LIN {X 0,Y 449.128,Z 238.43,A -85,B 0,C 180,E1 -8753.517,E2 -8753.517} C_VEL
LIN {X 0,Y 448.212,Z 232.343,A -85,B 0,C 180,E1 -8754.757,E2 -8754.757} C_VEL
LIN {X 0,Y 446.433,Z 223.879,A -85,B 0,C 180,E1 -8756.588,E2 -8756.588} C_VEL
LIN {X 0,Y 446.439,Z 223.874,A -85,B 0,C 180,E1 -8759.21,E2 -8759.21} C_VEL
LIN {X 0,Y 446.424,Z 223.875,A -85,B 0,C 180,E1 -8762.361,E2 -8762.361} C_VEL
LIN {X 0,Y 446.419,Z 223.88,A -85,B 0,C 180,E1 -8765.626,E2 -8765.626} C_VEL
LIN {X 0,Y 446.438,Z 223.874,A -85,B 0,C 180,E1 -8769.028,E2 -8769.028} C_VEL
LIN {X 0,Y 446.422,Z 223.874,A -85,B 0,C 180,E1 -8772.275,E2 -8772.275} C_VEL
LIN {X 0,Y 446.451,Z 223.873,A -85,B 0,C 180,E1 -8775.104,E2 -8775.104} C_VEL
LIN {X 0,Y 446.419,Z 223.874,A -85,B 0,C 180,E1 -8778.608,E2 -8778.608} C_VEL
LIN {X 0,Y 446.411,Z 223.875,A -85,B 0,C 180,E1 -8781.922,E2 -8781.922} C_VEL
LIN {X 0,Y 446.423,Z 223.877,A -85,B 0,C 180,E1 -8785.476,E2 -8785.476} C_VEL
LIN {X 0,Y 446.416,Z 223.874,A -85,B 0,C 180,E1 -8788.7,E2 -8788.7} C_VEL
LIN {X 0,Y 446.45,Z 223.873,A -85,B 0,C 180,E1 -8791.83,E2 -8791.83} C_VEL
LIN {X 0,Y 446.443,Z 223.867,A -85,B 0,C 180,E1 -8794.847,E2 -8794.847} C_VEL
LIN {X 0,Y 446.449,Z 223.867,A -85,B 0,C 180,E1 -8798.245,E2 -8798.245} C_VEL
LIN {X 0,Y 446.453,Z 223.873,A -85,B 0,C 180,E1 -8801.649,E2 -8801.649} C_VEL
LIN {X 0,Y 446.51,Z 223.86,A -85,B 0,C 180,E1 -8804.48,E2 -8804.48} C_VEL
LIN {X 0,Y 446.518,Z 223.857,A -85,B 0,C 180,E1 -8808.193,E2 -8808.193} C_VEL
LIN {X 0,Y 446.601,Z 223.849,A -85,B 0,C 180,E1 -8811.858,E2 -8811.858} C_VEL
LIN {X 0,Y 446.645,Z 223.843,A -85,B 0,C 180,E1 -8814.583,E2 -8814.583} C_VEL
LIN {X 0,Y 446.662,Z 223.838,A -85,B 0,C 180,E1 -8818.197,E2 -8818.197} C_VEL
LIN {X 0,Y 446.792,Z 223.828,A -85,B 0,C 180,E1 -8820,E2 -8820} C_VEL
LIN {X 0,Y 446.684,Z 223.837,A -85,B 0,C 180,E1 -8822.706,E2 -8822.706} C_VEL
LIN {X 0,Y 446.621,Z 223.848,A -85,B 0,C 180,E1 -8826.324,E2 -8826.324} C_VEL
LIN {X 0,Y 446.521,Z 223.862,A -85,B 0,C 180,E1 -8829.97,E2 -8829.97} C_VEL
LIN {X 0,Y 446.523,Z 223.859,A -85,B 0,C 180,E1 -8832.73,E2 -8832.73} C_VEL
LIN {X 0,Y 446.49,Z 223.863,A -85,B 0,C 180,E1 -8836.459,E2 -8836.459} C_VEL
LIN {X 0,Y 446.469,Z 223.869,A -85,B 0,C 180,E1 -8839.303,E2 -8839.303} C_VEL
LIN {X 0,Y 446.419,Z 223.868,A -85,B 0,C 180,E1 -8842.2,E2 -8842.2} C_VEL
LIN {X 0,Y 446.438,Z 223.875,A -85,B 0,C 180,E1 -8845.154,E2 -8845.154} C_VEL
LIN {X 0,Y 446.486,Z 223.865,A -85,B 0,C 180,E1 -8848.179,E2 -8848.179} C_VEL
LIN {X 0,Y 446.421,Z 223.876,A -85,B 0,C 180,E1 -8851.775,E2 -8851.775} C_VEL
LIN {X 0,Y 446.43,Z 223.872,A -85,B 0,C 180,E1 -8854.523,E2 -8854.523} C_VEL
LIN {X 0,Y 446.413,Z 223.875,A -85,B 0,C 180,E1 -8858.079,E2 -8858.079} C_VEL
LIN {X 0,Y 446.424,Z 223.875,A -85,B 0,C 180,E1 -8860.917,E2 -8860.917} C_VEL
LIN {X 0,Y 446.4,Z 223.88,A -85,B 0,C 180,E1 -8863.846,E2 -8863.846} C_VEL
LIN {X 0,Y 446.399,Z 223.873,A -85,B 0,C 180,E1 -8866.404,E2 -8866.404} C_VEL
LIN {X 0,Y 446.424,Z 223.88,A -85,B 0,C 180,E1 -8869.083,E2 -8869.083} C_VEL
LIN {X 0,Y 446.409,Z 223.879,A -85,B 0,C 180,E1 -8872.121,E2 -8872.121} C_VEL
LIN {X 0,Y 446.425,Z 223.88,A -85,B 0,C 180,E1 -8875.477,E2 -8875.477} C_VEL
LIN {X 0,Y 446.418,Z 223.875,A -85,B 0,C 180,E1 -8878.7,E2 -8878.7} C_VEL
LIN {X 0,Y 446.51,Z 224.034,A -85,B 0,C 180,E1 -8881.593,E2 -8881.593} C_VEL
LIN {X 0,Y 448.013,Z 232.082,A -85,B 0,C 180,E1 -8883.402,E2 -8883.402} C_VEL
LIN {X 0,Y 448.041,Z 238.215,A -85,B 0,C 180,E1 -8884.694,E2 -8884.694} C_VEL
LIN {X 0,Y 447.875,Z 245.014,A -85,B 0,C 180,E1 -8886.054,E2 -8886.054} C_VEL
LIN {X 0,Y 451.383,Z 262.204,A -85,B 0,C 180,E1 -8886.5,E2 -8886.5} C_VEL
LIN {X 0,Y 450.423,Z 352.698,A -85,B 0,C 180,E1 -8887.978,E2 -8887.978} C_VEL
LIN {X 0,Y 450.091,Z 365.924,A -85,B 0,C 180,E1 -8888.383,E2 -8888.383} C_VEL
LIN {X 0,Y 449.72,Z 376.471,A -85,B 0,C 180,E1 -8888.85,E2 -8888.85} C_VEL
LIN {X 0,Y 448.931,Z 381.929,A -85,B 0,C 180,E1 -8889.122,E2 -8889.122} C_VEL
LIN {X 0,Y 445.795,Z 390.661,A -85,B 0,C 180,E1 -8889.572,E2 -8889.572} C_VEL
LIN {X 0,Y 442.492,Z 399.015,A -85,B 0,C 180,E1 -8890.115,E2 -8890.115} C_VEL
LIN {X 0,Y 441.451,Z 403.881,A -85,B 0,C 180,E1 -8890.529,E2 -8890.529} C_VEL
LIN {X 0,Y 440.792,Z 414.392,A -85,B 0,C 180,E1 -8891.646,E2 -8891.646} C_VEL
LIN {X 0,Y 440.171,Z 423.362,A -85,B 0,C 180,E1 -8892.82,E2 -8892.82} C_VEL
LIN {X 0,Y 439.577,Z 432.067,A -85,B 0,C 180,E1 -8894.229,E2 -8894.229} C_VEL
LIN {X 0,Y 439.132,Z 438.983,A -85,B 0,C 180,E1 -8895.637,E2 -8895.637} C_VEL
LIN {X 0,Y 438.854,Z 444.496,A -85,B 0,C 180,E1 -8897.044,E2 -8897.044} C_VEL
LIN {X 0,Y 438.592,Z 448.795,A -85,B 0,C 180,E1 -8898.445,E2 -8898.445} C_VEL
LIN {X 0,Y 438.365,Z 452.009,A -85,B 0,C 180,E1 -8899.842,E2 -8899.842} C_VEL
LIN {X 0,Y 438.31,Z 453.6,A -85,B 0,C 180,E1 -8900.773,E2 -8900.773} C_VEL
LIN {X 0,Y 438.284,Z 454.779,A -85,B 0,C 180,E1 -8901.702,E2 -8901.702} C_VEL
LIN {X 0,Y 438.317,Z 455.855,A -85,B 0,C 180,E1 -8903.556,E2 -8903.556} C_VEL
LIN {X 0,Y 438.301,Z 455.817,A -85,B 0,C 180,E1 -8904.479,E2 -8904.479} C_VEL
LIN {X 0,Y 438.283,Z 455.391,A -85,B 0,C 180,E1 -8905.401,E2 -8905.401} C_VEL
LIN {X 0,Y 438.386,Z 453.275,A -85,B 0,C 180,E1 -8907.243,E2 -8907.243} C_VEL
LIN {X 0,Y 438.429,Z 450.625,A -85,B 0,C 180,E1 -8908.622,E2 -8908.622} C_VEL
LIN {X 0,Y 438.473,Z 446.978,A -85,B 0,C 180,E1 -8910,E2 -8910} C_VEL
LIN {X 0,Y 438.71,Z 442.223,A -85,B 0,C 180,E1 -8911.377,E2 -8911.377} C_VEL
LIN {X 0,Y 438.989,Z 436.231,A -85,B 0,C 180,E1 -8912.753,E2 -8912.753} C_VEL
LIN {X 0,Y 439.44,Z 428.782,A -85,B 0,C 180,E1 -8914.127,E2 -8914.127} C_VEL
LIN {X 0,Y 439.966,Z 421.176,A -85,B 0,C 180,E1 -8915.27,E2 -8915.27} C_VEL
LIN {X 0,Y 440.556,Z 411.939,A -85,B 0,C 180,E1 -8916.411,E2 -8916.411} C_VEL
LIN {X 0,Y 441.19,Z 401.671,A -85,B 0,C 180,E1 -8917.437,E2 -8917.437} C_VEL
LIN {X 0,Y 441.727,Z 390.301,A -85,B 0,C 180,E1 -8918.348,E2 -8918.348} C_VEL
LIN {X 0,Y 442.249,Z 378.407,A -85,B 0,C 180,E1 -8919.086,E2 -8919.086} C_VEL
LIN {X 0,Y 442.701,Z 365.181,A -85,B 0,C 180,E1 -8919.682,E2 -8919.682} C_VEL
LIN {X 0,Y 443.009,Z 351.886,A -85,B 0,C 180,E1 -8920.08,E2 -8920.08} C_VEL
LIN {X 0,Y 443.884,Z 263.104,A -85,B 0,C 180,E1 -8921.531,E2 -8921.531} C_VEL
LIN {X 0,Y 440.559,Z 244.83,A -85,B 0,C 180,E1 -8921.969,E2 -8921.969} C_VEL
LIN {X 0,Y 440.865,Z 232.497,A -85,B 0,C 180,E1 -8924.541,E2 -8924.541} C_VEL
LIN {X 0,Y 439.464,Z 224.747,A -85,B 0,C 180,E1 -8926.284,E2 -8926.284} C_VEL
LIN {X 0,Y 439.405,Z 224.747,A -85,B 0,C 180,E1 -8929.626,E2 -8929.626} C_VEL
LIN {X 0,Y 439.367,Z 224.757,A -85,B 0,C 180,E1 -8932.575,E2 -8932.575} C_VEL
LIN {X 0,Y 439.383,Z 224.749,A -85,B 0,C 180,E1 -8935.586,E2 -8935.586} C_VEL
LIN {X 0,Y 439.403,Z 224.755,A -85,B 0,C 180,E1 -8938.674,E2 -8938.674} C_VEL
LIN {X 0,Y 439.373,Z 224.751,A -85,B 0,C 180,E1 -8942.03,E2 -8942.03} C_VEL
LIN {X 0,Y 439.396,Z 224.748,A -85,B 0,C 180,E1 -8945.34,E2 -8945.34} C_VEL
LIN {X 0,Y 439.379,Z 224.756,A -85,B 0,C 180,E1 -8948.595,E2 -8948.595} C_VEL
LIN {X 0,Y 439.39,Z 224.749,A -85,B 0,C 180,E1 -8951.256,E2 -8951.256} C_VEL
LIN {X 0,Y 439.401,Z 224.754,A -85,B 0,C 180,E1 -8954.729,E2 -8954.729} C_VEL
LIN {X 0,Y 439.385,Z 224.749,A -85,B 0,C 180,E1 -8957.794,E2 -8957.794} C_VEL
LIN {X 0,Y 439.396,Z 224.75,A -85,B 0,C 180,E1 -8960.224,E2 -8960.224} C_VEL
LIN {X 0,Y 439.373,Z 224.75,A -85,B 0,C 180,E1 -8963.712,E2 -8963.712} C_VEL
LIN {X 0,Y 439.374,Z 224.753,A -85,B 0,C 180,E1 -8967.054,E2 -8967.054} C_VEL
LIN {X 0,Y 439.383,Z 224.752,A -85,B 0,C 180,E1 -8970.274,E2 -8970.274} C_VEL
LIN {X 0,Y 439.42,Z 224.745,A -85,B 0,C 180,E1 -8973.395,E2 -8973.395} C_VEL
LIN {X 0,Y 439.383,Z 224.754,A -85,B 0,C 180,E1 -8976.429,E2 -8976.429} C_VEL
LIN {X 0,Y 439.389,Z 224.749,A -85,B 0,C 180,E1 -8979.397,E2 -8979.397} C_VEL
LIN {X 0,Y 439.405,Z 224.75,A -85,B 0,C 180,E1 -8982.308,E2 -8982.308} C_VEL
LIN {X 0,Y 439.446,Z 224.743,A -85,B 0,C 180,E1 -8985.174,E2 -8985.174} C_VEL
LIN {X 0,Y 439.484,Z 224.738,A -85,B 0,C 180,E1 -8988.001,E2 -8988.001} C_VEL
LIN {X 0,Y 439.504,Z 224.734,A -85,B 0,C 180,E1 -8991.725,E2 -8991.725} C_VEL
LIN {X 0,Y 439.611,Z 224.727,A -85,B 0,C 180,E1 -8994.496,E2 -8994.496} C_VEL
LIN {X 0,Y 439.636,Z 224.72,A -85,B 0,C 180,E1 -8998.168,E2 -8998.168} C_VEL
LIN {X 0,Y 439.761,Z 224.703,A -85,B 0,C 180,E1 -9000,E2 -9000} C_VEL
LIN {X 0,Y 439.633,Z 224.724,A -85,B 0,C 180,E1 -9002.749,E2 -9002.749} C_VEL
LIN {X 0,Y 439.618,Z 224.725,A -85,B 0,C 180,E1 -9006.425,E2 -9006.425} C_VEL
LIN {X 0,Y 439.499,Z 224.736,A -85,B 0,C 180,E1 -9009.202,E2 -9009.202} C_VEL
LIN {X 0,Y 439.466,Z 224.742,A -85,B 0,C 180,E1 -9012.938,E2 -9012.938} C_VEL
LIN {X 0,Y 439.447,Z 224.746,A -85,B 0,C 180,E1 -9016.348,E2 -9016.348} C_VEL
LIN {X 0,Y 439.402,Z 224.746,A -85,B 0,C 180,E1 -9019.626,E2 -9019.626} C_VEL
LIN {X 0,Y 439.365,Z 224.759,A -85,B 0,C 180,E1 -9022.575,E2 -9022.575} C_VEL
LIN {X 0,Y 439.381,Z 224.749,A -85,B 0,C 180,E1 -9025.586,E2 -9025.586} C_VEL
LIN {X 0,Y 439.4,Z 224.753,A -85,B 0,C 180,E1 -9028.675,E2 -9028.675} C_VEL
LIN {X 0,Y 439.369,Z 224.752,A -85,B 0,C 180,E1 -9032.03,E2 -9032.03} C_VEL
LIN {X 0,Y 439.391,Z 224.748,A -85,B 0,C 180,E1 -9035.34,E2 -9035.34} C_VEL
LIN {X 0,Y 439.363,Z 224.759,A -85,B 0,C 180,E1 -9038.597,E2 -9038.597} C_VEL
LIN {X 0,Y 439.381,Z 224.75,A -85,B 0,C 180,E1 -9041.256,E2 -9041.256} C_VEL
LIN {X 0,Y 439.399,Z 224.753,A -85,B 0,C 180,E1 -9044.73,E2 -9044.73} C_VEL
LIN {X 0,Y 439.385,Z 224.749,A -85,B 0,C 180,E1 -9047.794,E2 -9047.794} C_VEL
LIN {X 0,Y 439.394,Z 224.751,A -85,B 0,C 180,E1 -9050.224,E2 -9050.224} C_VEL
LIN {X 0,Y 439.373,Z 224.75,A -85,B 0,C 180,E1 -9053.713,E2 -9053.713} C_VEL
LIN {X 0,Y 439.373,Z 224.752,A -85,B 0,C 180,E1 -9057.054,E2 -9057.054} C_VEL
LIN {X 0,Y 439.383,Z 224.754,A -85,B 0,C 180,E1 -9060.274,E2 -9060.274} C_VEL
LIN {X 0,Y 439.42,Z 224.75,A -85,B 0,C 180,E1 -9063.396,E2 -9063.396} C_VEL
LIN {X 0,Y 439.438,Z 224.842,A -85,B 0,C 180,E1 -9063.812,E2 -9063.812} C_VEL
LIN {X 0,Y 441.714,Z 237.096,A -85,B 0,C 180,E1 -9066.313,E2 -9066.313} C_VEL
LIN {X 0,Y 441.117,Z 251.239,A -85,B 0,C 180,E1 -9068.993,E2 -9068.993} C_VEL
LIN {X 0,Y 440.279,Z 267.688,A -85,B 0,C 180,E1 -9072.061,E2 -9072.061} C_VEL
LIN {X 0,Y 443.65,Z 290.825,A -85,B 0,C 180,E1 -9072.567,E2 -9072.567} C_VEL
LIN {X 0,Y 442.927,Z 376.061,A -85,B 0,C 180,E1 -9073.967,E2 -9073.967} C_VEL
LIN {X 0,Y 442.438,Z 389.288,A -85,B 0,C 180,E1 -9074.363,E2 -9074.363} C_VEL
LIN {X 0,Y 441.929,Z 401.448,A -85,B 0,C 180,E1 -9074.906,E2 -9074.906} C_VEL
LIN {X 0,Y 441.415,Z 412.909,A -85,B 0,C 180,E1 -9075.595,E2 -9075.595} C_VEL
LIN {X 0,Y 440.76,Z 423.999,A -85,B 0,C 180,E1 -9076.454,E2 -9076.454} C_VEL
LIN {X 0,Y 440.193,Z 435.24,A -85,B 0,C 180,E1 -9077.553,E2 -9077.553} C_VEL
LIN {X 0,Y 439.685,Z 444.751,A -85,B 0,C 180,E1 -9078.708,E2 -9078.708} C_VEL
LIN {X 0,Y 439.149,Z 453.898,A -85,B 0,C 180,E1 -9080.094,E2 -9080.094} C_VEL
LIN {X 0,Y 438.795,Z 461.267,A -85,B 0,C 180,E1 -9081.48,E2 -9081.48} C_VEL
LIN {X 0,Y 438.495,Z 468.015,A -85,B 0,C 180,E1 -9083.096,E2 -9083.096} C_VEL
LIN {X 0,Y 438.377,Z 472.466,A -85,B 0,C 180,E1 -9084.48,E2 -9084.48} C_VEL
LIN {X 0,Y 438.34,Z 474.814,A -85,B 0,C 180,E1 -9085.402,E2 -9085.402} C_VEL
LIN {X 0,Y 438.28,Z 476.73,A -85,B 0,C 180,E1 -9086.322,E2 -9086.322} C_VEL
LIN {X 0,Y 438.34,Z 478.209,A -85,B 0,C 180,E1 -9087.243,E2 -9087.243} C_VEL
LIN {X 0,Y 438.252,Z 479.891,A -85,B 0,C 180,E1 -9089.081,E2 -9089.081} C_VEL
LIN {X 0,Y 438.254,Z 480.153,A -85,B 0,C 180,E1 -9090,E2 -9090} C_VEL
LIN {X 0,Y 438.252,Z 480.01,A -85,B 0,C 180,E1 -9090.919,E2 -9090.919} C_VEL
LIN {X 0,Y 438.34,Z 478.489,A -85,B 0,C 180,E1 -9092.757,E2 -9092.757} C_VEL
LIN {X 0,Y 438.279,Z 477.139,A -85,B 0,C 180,E1 -9093.678,E2 -9093.678} C_VEL
LIN {X 0,Y 438.382,Z 474.292,A -85,B 0,C 180,E1 -9095.059,E2 -9095.059} C_VEL
LIN {X 0,Y 438.448,Z 470.421,A -85,B 0,C 180,E1 -9096.442,E2 -9096.442} C_VEL
LIN {X 0,Y 438.685,Z 465.432,A -85,B 0,C 180,E1 -9097.827,E2 -9097.827} C_VEL
LIN {X 0,Y 438.989,Z 459.173,A -85,B 0,C 180,E1 -9099.212,E2 -9099.212} C_VEL
LIN {X 0,Y 439.456,Z 451.355,A -85,B 0,C 180,E1 -9100.598,E2 -9100.598} C_VEL
LIN {X 0,Y 440.188,Z 441.612,A -85,B 0,C 180,E1 -9101.979,E2 -9101.979} C_VEL
LIN {X 0,Y 440.904,Z 431.224,A -85,B 0,C 180,E1 -9103.159,E2 -9103.159} C_VEL
LIN {X 0,Y 441.378,Z 421.543,A -85,B 0,C 180,E1 -9104.053,E2 -9104.053} C_VEL
LIN {X 0,Y 442.056,Z 410.696,A -85,B 0,C 180,E1 -9104.854,E2 -9104.854} C_VEL
LIN {X 0,Y 442.696,Z 398.737,A -85,B 0,C 180,E1 -9105.539,E2 -9105.539} C_VEL
LIN {X 0,Y 443.289,Z 385.693,A -85,B 0,C 180,E1 -9106.078,E2 -9106.078} C_VEL
LIN {X 0,Y 443.66,Z 372.689,A -85,B 0,C 180,E1 -9106.419,E2 -9106.419} C_VEL
LIN {X 0,Y 444.426,Z 289.513,A -85,B 0,C 180,E1 -9107.788,E2 -9107.788} C_VEL
LIN {X 0,Y 440.628,Z 267.417,A -85,B 0,C 180,E1 -9108.352,E2 -9108.352} C_VEL
LIN {X 0,Y 441.566,Z 250.995,A -85,B 0,C 180,E1 -9111.473,E2 -9111.473} C_VEL
LIN {X 0,Y 442.212,Z 239.66,A -85,B 0,C 180,E1 -9113.659,E2 -9113.659} C_VEL
LIN {X 0,Y 440.893,Z 231.848,A -85,B 0,C 180,E1 -9115.29,E2 -9115.29} C_VEL
LIN {X 0,Y 439.412,Z 224.754,A -85,B 0,C 180,E1 -9116.861,E2 -9116.861} C_VEL
LIN {X 0,Y 439.378,Z 224.752,A -85,B 0,C 180,E1 -9119.726,E2 -9119.726} C_VEL
LIN {X 0,Y 439.374,Z 224.755,A -85,B 0,C 180,E1 -9122.946,E2 -9122.946} C_VEL
LIN {X 0,Y 439.373,Z 224.752,A -85,B 0,C 180,E1 -9126.287,E2 -9126.287} C_VEL
LIN {X 0,Y 439.403,Z 224.752,A -85,B 0,C 180,E1 -9129.849,E2 -9129.849} C_VEL
LIN {X 0,Y 439.371,Z 224.753,A -85,B 0,C 180,E1 -9132.625,E2 -9132.625} C_VEL
LIN {X 0,Y 439.399,Z 224.753,A -85,B 0,C 180,E1 -9135.27,E2 -9135.27} C_VEL
LIN {X 0,Y 439.382,Z 224.751,A -85,B 0,C 180,E1 -9138.744,E2 -9138.744} C_VEL
LIN {X 0,Y 439.365,Z 224.757,A -85,B 0,C 180,E1 -9141.609,E2 -9141.609} C_VEL
LIN {X 0,Y 439.396,Z 224.749,A -85,B 0,C 180,E1 -9144.844,E2 -9144.844} C_VEL
LIN {X 0,Y 439.373,Z 224.752,A -85,B 0,C 180,E1 -9148.139,E2 -9148.139} C_VEL
LIN {X 0,Y 439.41,Z 224.752,A -85,B 0,C 180,E1 -9151.604,E2 -9151.604} C_VEL
LIN {X 0,Y 439.38,Z 224.746,A -85,B 0,C 180,E1 -9154.414,E2 -9154.414} C_VEL
LIN {X 0,Y 439.365,Z 224.758,A -85,B 0,C 180,E1 -9157.425,E2 -9157.425} C_VEL
LIN {X 0,Y 439.442,Z 224.743,A -85,B 0,C 180,E1 -9160.663,E2 -9160.663} C_VEL
LIN {X 0,Y 439.464,Z 224.738,A -85,B 0,C 180,E1 -9164.225,E2 -9164.225} C_VEL
LIN {X 0,Y 439.484,Z 224.734,A -85,B 0,C 180,E1 -9168.001,E2 -9168.001} C_VEL
LIN {X 0,Y 439.549,Z 224.729,A -85,B 0,C 180,E1 -9171.726,E2 -9171.726} C_VEL
LIN {X 0,Y 439.621,Z 224.718,A -85,B 0,C 180,E1 -9174.496,E2 -9174.496} C_VEL
LIN {X 0,Y 439.632,Z 224.714,A -85,B 0,C 180,E1 -9178.168,E2 -9178.168} C_VEL
LIN {X 0,Y 439.762,Z 224.704,A -85,B 0,C 180,E1 -9180,E2 -9180} C_VEL
LIN {X 0,Y 439.633,Z 224.716,A -85,B 0,C 180,E1 -9182.749,E2 -9182.749} C_VEL
LIN {X 0,Y 439.586,Z 224.724,A -85,B 0,C 180,E1 -9186.487,E2 -9186.487} C_VEL
LIN {X 0,Y 439.496,Z 224.735,A -85,B 0,C 180,E1 -9189.202,E2 -9189.202} C_VEL
LIN {X 0,Y 439.466,Z 224.739,A -85,B 0,C 180,E1 -9192.938,E2 -9192.938} C_VEL
LIN {X 0,Y 439.447,Z 224.741,A -85,B 0,C 180,E1 -9196.348,E2 -9196.348} C_VEL
LIN {X 0,Y 439.403,Z 224.751,A -85,B 0,C 180,E1 -9199.626,E2 -9199.626} C_VEL
LIN {X 0,Y 439.364,Z 224.747,A -85,B 0,C 180,E1 -9202.576,E2 -9202.576} C_VEL
LIN {X 0,Y 439.387,Z 224.75,A -85,B 0,C 180,E1 -9205.586,E2 -9205.586} C_VEL
LIN {X 0,Y 439.418,Z 224.746,A -85,B 0,C 180,E1 -9208.674,E2 -9208.674} C_VEL
LIN {X 0,Y 439.372,Z 224.752,A -85,B 0,C 180,E1 -9212.031,E2 -9212.031} C_VEL
LIN {X 0,Y 439.395,Z 224.755,A -85,B 0,C 180,E1 -9215.34,E2 -9215.34} C_VEL
LIN {X 0,Y 439.376,Z 224.751,A -85,B 0,C 180,E1 -9218.596,E2 -9218.596} C_VEL
LIN {X 0,Y 439.383,Z 224.755,A -85,B 0,C 180,E1 -9221.256,E2 -9221.256} C_VEL
LIN {X 0,Y 439.4,Z 224.75,A -85,B 0,C 180,E1 -9224.73,E2 -9224.73} C_VEL
LIN {X 0,Y 439.386,Z 224.757,A -85,B 0,C 180,E1 -9227.794,E2 -9227.794} C_VEL
LIN {X 0,Y 439.36,Z 224.754,A -85,B 0,C 180,E1 -9230.22,E2 -9230.22} C_VEL
LIN {X 0,Y 439.375,Z 224.759,A -85,B 0,C 180,E1 -9233.713,E2 -9233.713} C_VEL
LIN {X 0,Y 439.374,Z 224.757,A -85,B 0,C 180,E1 -9237.054,E2 -9237.054} C_VEL
LIN {X 0,Y 439.413,Z 224.746,A -85,B 0,C 180,E1 -9240.803,E2 -9240.803} C_VEL
LIN {X 0,Y 439.469,Z 224.866,A -85,B 0,C 180,E1 -9241.33,E2 -9241.33} C_VEL
LIN {X 0,Y 441.176,Z 234.455,A -85,B 0,C 180,E1 -9243.51,E2 -9243.51} C_VEL
LIN {X 0,Y 440.928,Z 244.858,A -85,B 0,C 180,E1 -9245.706,E2 -9245.706} C_VEL
LIN {X 0,Y 444.698,Z 263.061,A -85,B 0,C 180,E1 -9246.209,E2 -9246.209} C_VEL
LIN {X 0,Y 443.694,Z 352.439,A -85,B 0,C 180,E1 -9247.687,E2 -9247.687} C_VEL
LIN {X 0,Y 443.334,Z 365.811,A -85,B 0,C 180,E1 -9248.097,E2 -9248.097} C_VEL
LIN {X 0,Y 442.882,Z 378.054,A -85,B 0,C 180,E1 -9248.655,E2 -9248.655} C_VEL
LIN {X 0,Y 442.28,Z 390.342,A -85,B 0,C 180,E1 -9249.416,E2 -9249.416} C_VEL
LIN {X 0,Y 441.637,Z 401.326,A -85,B 0,C 180,E1 -9250.297,E2 -9250.297} C_VEL
LIN {X 0,Y 441.451,Z 403.881,A -85,B 0,C 180,E1 -9250.529,E2 -9250.529} C_VEL
LIN {X 0,Y 440.432,Z 408.624,A -85,B 0,C 180,E1 -9250.973,E2 -9250.973} C_VEL
LIN {X 0,Y 435.711,Z 418.906,A -85,B 0,C 180,E1 -9252.034,E2 -9252.034} C_VEL
LIN {X 0,Y 433.495,Z 424.327,A -85,B 0,C 180,E1 -9252.731,E2 -9252.731} C_VEL
LIN {X 0,Y 433.028,Z 426.865,A -85,B 0,C 180,E1 -9253.118,E2 -9253.118} C_VEL
LIN {X 0,Y 432.459,Z 434.376,A -85,B 0,C 180,E1 -9254.446,E2 -9254.446} C_VEL
LIN {X 0,Y 432.039,Z 440.901,A -85,B 0,C 180,E1 -9255.877,E2 -9255.877} C_VEL
LIN {X 0,Y 431.719,Z 446.054,A -85,B 0,C 180,E1 -9257.305,E2 -9257.305} C_VEL
LIN {X 0,Y 431.452,Z 450.032,A -85,B 0,C 180,E1 -9258.728,E2 -9258.728} C_VEL
LIN {X 0,Y 431.317,Z 452.07,A -85,B 0,C 180,E1 -9259.675,E2 -9259.675} C_VEL
LIN {X 0,Y 431.187,Z 454.899,A -85,B 0,C 180,E1 -9261.565,E2 -9261.565} C_VEL
LIN {X 0,Y 431.211,Z 455.672,A -85,B 0,C 180,E1 -9262.508,E2 -9262.508} C_VEL
LIN {X 0,Y 431.248,Z 456.094,A -85,B 0,C 180,E1 -9263.782,E2 -9263.782} C_VEL
LIN {X 0,Y 431.207,Z 455.63,A -85,B 0,C 180,E1 -9265.326,E2 -9265.326} C_VEL
LIN {X 0,Y 431.177,Z 454.814,A -85,B 0,C 180,E1 -9266.262,E2 -9266.262} C_VEL
LIN {X 0,Y 431.291,Z 453.582,A -85,B 0,C 180,E1 -9267.198,E2 -9267.198} C_VEL
LIN {X 0,Y 431.329,Z 450.982,A -85,B 0,C 180,E1 -9268.599,E2 -9268.599} C_VEL
LIN {X 0,Y 431.405,Z 447.388,A -85,B 0,C 180,E1 -9270,E2 -9270} C_VEL
LIN {X 0,Y 431.63,Z 442.691,A -85,B 0,C 180,E1 -9271.399,E2 -9271.399} C_VEL
LIN {X 0,Y 431.929,Z 436.76,A -85,B 0,C 180,E1 -9272.798,E2 -9272.798} C_VEL
LIN {X 0,Y 432.393,Z 429.381,A -85,B 0,C 180,E1 -9274.194,E2 -9274.194} C_VEL
LIN {X 0,Y 432.936,Z 421.856,A -85,B 0,C 180,E1 -9275.356,E2 -9275.356} C_VEL
LIN {X 0,Y 433.559,Z 412.752,A -85,B 0,C 180,E1 -9276.515,E2 -9276.515} C_VEL
LIN {X 0,Y 434.184,Z 402.633,A -85,B 0,C 180,E1 -9277.557,E2 -9277.557} C_VEL
LIN {X 0,Y 434.761,Z 391.43,A -85,B 0,C 180,E1 -9278.482,E2 -9278.482} C_VEL
LIN {X 0,Y 435.283,Z 380.802,A -85,B 0,C 180,E1 -9279.174,E2 -9279.174} C_VEL
LIN {X 0,Y 435.764,Z 367.919,A -85,B 0,C 180,E1 -9279.808,E2 -9279.808} C_VEL
LIN {X 0,Y 436.042,Z 354.598,A -85,B 0,C 180,E1 -9280.248,E2 -9280.248} C_VEL
LIN {X 0,Y 436.422,Z 330.852,A -85,B 0,C 180,E1 -9280.675,E2 -9280.675} C_VEL
LIN {X 0,Y 436.959,Z 263.114,A -85,B 0,C 180,E1 -9281.79,E2 -9281.79} C_VEL
LIN {X 0,Y 433.621,Z 244.924,A -85,B 0,C 180,E1 -9282.252,E2 -9282.252} C_VEL
LIN {X 0,Y 433.936,Z 234.094,A -85,B 0,C 180,E1 -9284.539,E2 -9284.539} C_VEL
LIN {X 0,Y 432.412,Z 225.625,A -85,B 0,C 180,E1 -9286.477,E2 -9286.477} C_VEL
LIN {X 0,Y 432.342,Z 225.627,A -85,B 0,C 180,E1 -9289.96,E2 -9289.96} C_VEL
LIN {X 0,Y 432.321,Z 225.633,A -85,B 0,C 180,E1 -9292.964,E2 -9292.964} C_VEL
LIN {X 0,Y 432.342,Z 225.63,A -85,B 0,C 180,E1 -9295.002,E2 -9295.002} C_VEL
LIN {X 0,Y 432.35,Z 225.627,A -85,B 0,C 180,E1 -9298.126,E2 -9298.126} C_VEL
LIN {X 0,Y 432.323,Z 225.629,A -85,B 0,C 180,E1 -9301.346,E2 -9301.346} C_VEL
LIN {X 0,Y 432.342,Z 225.634,A -85,B 0,C 180,E1 -9304.677,E2 -9304.677} C_VEL
LIN {X 0,Y 432.338,Z 225.628,A -85,B 0,C 180,E1 -9308.15,E2 -9308.15} C_VEL
LIN {X 0,Y 432.334,Z 225.627,A -85,B 0,C 180,E1 -9311.602,E2 -9311.602} C_VEL
LIN {X 0,Y 432.335,Z 225.631,A -85,B 0,C 180,E1 -9314.347,E2 -9314.347} C_VEL
LIN {X 0,Y 432.318,Z 225.632,A -85,B 0,C 180,E1 -9317.016,E2 -9317.016} C_VEL
LIN {X 0,Y 432.333,Z 225.627,A -85,B 0,C 180,E1 -9319.821,E2 -9319.821} C_VEL
LIN {X 0,Y 432.306,Z 225.634,A -85,B 0,C 180,E1 -9323.022,E2 -9323.022} C_VEL
LIN {X 0,Y 432.36,Z 225.625,A -85,B 0,C 180,E1 -9325.996,E2 -9325.996} C_VEL
LIN {X 0,Y 432.349,Z 225.625,A -85,B 0,C 180,E1 -9329.489,E2 -9329.489} C_VEL
LIN {X 0,Y 432.386,Z 225.625,A -85,B 0,C 180,E1 -9332.928,E2 -9332.928} C_VEL
LIN {X 0,Y 432.366,Z 225.624,A -85,B 0,C 180,E1 -9336.023,E2 -9336.023} C_VEL
LIN {X 0,Y 432.351,Z 225.628,A -85,B 0,C 180,E1 -9339.046,E2 -9339.046} C_VEL
LIN {X 0,Y 432.361,Z 225.625,A -85,B 0,C 180,E1 -9342.01,E2 -9342.01} C_VEL
LIN {X 0,Y 432.394,Z 225.624,A -85,B 0,C 180,E1 -9344.926,E2 -9344.926} C_VEL
LIN {X 0,Y 432.46,Z 225.612,A -85,B 0,C 180,E1 -9347.803,E2 -9347.803} C_VEL
LIN {X 0,Y 432.464,Z 225.611,A -85,B 0,C 180,E1 -9351.59,E2 -9351.59} C_VEL
LIN {X 0,Y 432.586,Z 225.601,A -85,B 0,C 180,E1 -9354.406,E2 -9354.406} C_VEL
LIN {X 0,Y 432.605,Z 225.596,A -85,B 0,C 180,E1 -9358.138,E2 -9358.138} C_VEL
LIN {X 0,Y 432.731,Z 225.579,A -85,B 0,C 180,E1 -9360,E2 -9360} C_VEL
LIN {X 0,Y 432.585,Z 225.601,A -85,B 0,C 180,E1 -9362.794,E2 -9362.794} C_VEL
LIN {X 0,Y 432.573,Z 225.604,A -85,B 0,C 180,E1 -9366.53,E2 -9366.53} C_VEL
LIN {X 0,Y 432.442,Z 225.614,A -85,B 0,C 180,E1 -9369.353,E2 -9369.353} C_VEL
LIN {X 0,Y 432.432,Z 225.62,A -85,B 0,C 180,E1 -9372.803,E2 -9372.803} C_VEL
LIN {X 0,Y 432.412,Z 225.624,A -85,B 0,C 180,E1 -9376.478,E2 -9376.478} C_VEL
LIN {X 0,Y 432.339,Z 225.628,A -85,B 0,C 180,E1 -9379.96,E2 -9379.96} C_VEL
LIN {X 0,Y 432.318,Z 225.632,A -85,B 0,C 180,E1 -9382.964,E2 -9382.964} C_VEL
LIN {X 0,Y 432.34,Z 225.629,A -85,B 0,C 180,E1 -9385.002,E2 -9385.002} C_VEL
LIN {X 0,Y 432.347,Z 225.628,A -85,B 0,C 180,E1 -9388.126,E2 -9388.126} C_VEL
LIN {X 0,Y 432.321,Z 225.629,A -85,B 0,C 180,E1 -9391.346,E2 -9391.346} C_VEL
LIN {X 0,Y 432.337,Z 225.633,A -85,B 0,C 180,E1 -9394.677,E2 -9394.677} C_VEL
LIN {X 0,Y 432.33,Z 225.63,A -85,B 0,C 180,E1 -9398.151,E2 -9398.151} C_VEL
LIN {X 0,Y 432.324,Z 225.628,A -85,B 0,C 180,E1 -9401.601,E2 -9401.601} C_VEL
LIN {X 0,Y 432.334,Z 225.632,A -85,B 0,C 180,E1 -9404.347,E2 -9404.347} C_VEL
LIN {X 0,Y 432.317,Z 225.631,A -85,B 0,C 180,E1 -9407.016,E2 -9407.016} C_VEL
LIN {X 0,Y 432.332,Z 225.628,A -85,B 0,C 180,E1 -9409.821,E2 -9409.821} C_VEL
LIN {X 0,Y 432.305,Z 225.633,A -85,B 0,C 180,E1 -9413.022,E2 -9413.022} C_VEL
LIN {X 0,Y 432.36,Z 225.626,A -85,B 0,C 180,E1 -9415.997,E2 -9415.997} C_VEL
LIN {X 0,Y 432.348,Z 225.626,A -85,B 0,C 180,E1 -9419.49,E2 -9419.49} C_VEL
LIN {X 0,Y 432.386,Z 225.628,A -85,B 0,C 180,E1 -9422.928,E2 -9422.928} C_VEL
LIN {X 0,Y 432.385,Z 225.677,A -85,B 0,C 180,E1 -9423.598,E2 -9423.598} C_VEL
LIN {X 0,Y 434.722,Z 238.008,A -85,B 0,C 180,E1 -9426.161,E2 -9426.161} C_VEL
LIN {X 0,Y 434.451,Z 247.022,A -85,B 0,C 180,E1 -9427.907,E2 -9427.907} C_VEL
LIN {X 0,Y 433.52,Z 263.68,A -85,B 0,C 180,E1 -9431.081,E2 -9431.081} C_VEL
LIN {X 0,Y 433.343,Z 267.461,A -85,B 0,C 180,E1 -9431.795,E2 -9431.795} C_VEL
LIN {X 0,Y 436.801,Z 290.927,A -85,B 0,C 180,E1 -9432.32,E2 -9432.32} C_VEL
LIN {X 0,Y 436.06,Z 375.899,A -85,B 0,C 180,E1 -9433.738,E2 -9433.738} C_VEL
LIN {X 0,Y 435.547,Z 389.116,A -85,B 0,C 180,E1 -9434.139,E2 -9434.139} C_VEL
LIN {X 0,Y 435.004,Z 401.841,A -85,B 0,C 180,E1 -9434.719,E2 -9434.719} C_VEL
LIN {X 0,Y 434.405,Z 413.932,A -85,B 0,C 180,E1 -9435.477,E2 -9435.477} C_VEL
LIN {X 0,Y 433.738,Z 425.182,A -85,B 0,C 180,E1 -9436.385,E2 -9436.385} C_VEL
LIN {X 0,Y 433.151,Z 435.863,A -85,B 0,C 180,E1 -9437.466,E2 -9437.466} C_VEL
LIN {X 0,Y 432.692,Z 444.354,A -85,B 0,C 180,E1 -9438.523,E2 -9438.523} C_VEL
LIN {X 0,Y 432.09,Z 453.542,A -85,B 0,C 180,E1 -9439.93,E2 -9439.93} C_VEL
LIN {X 0,Y 431.731,Z 460.94,A -85,B 0,C 180,E1 -9441.34,E2 -9441.34} C_VEL
LIN {X 0,Y 431.416,Z 467.725,A -85,B 0,C 180,E1 -9442.982,E2 -9442.982} C_VEL
LIN {X 0,Y 431.281,Z 472.198,A -85,B 0,C 180,E1 -9444.389,E2 -9444.389} C_VEL
LIN {X 0,Y 431.27,Z 474.558,A -85,B 0,C 180,E1 -9445.326,E2 -9445.326} C_VEL
LIN {X 0,Y 431.187,Z 476.483,A -85,B 0,C 180,E1 -9446.262,E2 -9446.262} C_VEL
LIN {X 0,Y 431.236,Z 477.98,A -85,B 0,C 180,E1 -9447.198,E2 -9447.198} C_VEL
LIN {X 0,Y 431.203,Z 479.026,A -85,B 0,C 180,E1 -9448.132,E2 -9448.132} C_VEL
LIN {X 0,Y 431.168,Z 479.952,A -85,B 0,C 180,E1 -9450,E2 -9450} C_VEL
LIN {X 0,Y 431.169,Z 479.826,A -85,B 0,C 180,E1 -9450.934,E2 -9450.934} C_VEL
LIN {X 0,Y 431.203,Z 479.269,A -85,B 0,C 180,E1 -9451.868,E2 -9451.868} C_VEL
LIN {X 0,Y 431.235,Z 478.324,A -85,B 0,C 180,E1 -9452.802,E2 -9452.802} C_VEL
LIN {X 0,Y 431.186,Z 476.983,A -85,B 0,C 180,E1 -9453.738,E2 -9453.738} C_VEL
LIN {X 0,Y 431.293,Z 474.155,A -85,B 0,C 180,E1 -9455.142,E2 -9455.142} C_VEL
LIN {X 0,Y 431.377,Z 470.305,A -85,B 0,C 180,E1 -9456.549,E2 -9456.549} C_VEL
LIN {X 0,Y 431.609,Z 465.339,A -85,B 0,C 180,E1 -9457.956,E2 -9457.956} C_VEL
LIN {X 0,Y 431.973,Z 459.106,A -85,B 0,C 180,E1 -9459.363,E2 -9459.363} C_VEL
LIN {X 0,Y 432.435,Z 451.333,A -85,B 0,C 180,E1 -9460.772,E2 -9460.772} C_VEL
LIN {X 0,Y 433.224,Z 441.626,A -85,B 0,C 180,E1 -9462.175,E2 -9462.175} C_VEL
LIN {X 0,Y 433.936,Z 432,A -85,B 0,C 180,E1 -9463.301,E2 -9463.301} C_VEL
LIN {X 0,Y 434.489,Z 421.691,A -85,B 0,C 180,E1 -9464.281,E2 -9464.281} C_VEL
LIN {X 0,Y 435.212,Z 410.93,A -85,B 0,C 180,E1 -9465.093,E2 -9465.093} C_VEL
LIN {X 0,Y 435.895,Z 399.093,A -85,B 0,C 180,E1 -9465.788,E2 -9465.788} C_VEL
LIN {X 0,Y 436.518,Z 386.338,A -85,B 0,C 180,E1 -9466.335,E2 -9466.335} C_VEL
LIN {X 0,Y 436.898,Z 373.975,A -85,B 0,C 180,E1 -9466.681,E2 -9466.681} C_VEL
LIN {X 0,Y 437.753,Z 290.469,A -85,B 0,C 180,E1 -9468.079,E2 -9468.079} C_VEL
LIN {X 0,Y 433.744,Z 267.152,A -85,B 0,C 180,E1 -9468.698,E2 -9468.698} C_VEL
LIN {X 0,Y 434.701,Z 250.966,A -85,B 0,C 180,E1 -9471.83,E2 -9471.83} C_VEL
LIN {X 0,Y 435.308,Z 240.895,A -85,B 0,C 180,E1 -9473.805,E2 -9473.805} C_VEL
LIN {X 0,Y 433.718,Z 232.083,A -85,B 0,C 180,E1 -9475.687,E2 -9475.687} C_VEL
LIN {X 0,Y 432.368,Z 225.631,A -85,B 0,C 180,E1 -9477.139,E2 -9477.139} C_VEL
LIN {X 0,Y 432.348,Z 225.629,A -85,B 0,C 180,E1 -9480.51,E2 -9480.51} C_VEL
LIN {X 0,Y 432.36,Z 225.627,A -85,B 0,C 180,E1 -9484.003,E2 -9484.003} C_VEL
LIN {X 0,Y 432.321,Z 225.635,A -85,B 0,C 180,E1 -9487.196,E2 -9487.196} C_VEL
LIN {X 0,Y 432.332,Z 225.63,A -85,B 0,C 180,E1 -9490.179,E2 -9490.179} C_VEL
LIN {X 0,Y 432.315,Z 225.634,A -85,B 0,C 180,E1 -9493.061,E2 -9493.061} C_VEL
LIN {X 0,Y 432.334,Z 225.633,A -85,B 0,C 180,E1 -9495.665,E2 -9495.665} C_VEL
LIN {X 0,Y 432.325,Z 225.63,A -85,B 0,C 180,E1 -9498.399,E2 -9498.399} C_VEL
LIN {X 0,Y 432.33,Z 225.63,A -85,B 0,C 180,E1 -9501.849,E2 -9501.849} C_VEL
LIN {X 0,Y 432.337,Z 225.633,A -85,B 0,C 180,E1 -9505.323,E2 -9505.323} C_VEL
LIN {X 0,Y 432.321,Z 225.63,A -85,B 0,C 180,E1 -9508.654,E2 -9508.654} C_VEL
LIN {X 0,Y 432.348,Z 225.629,A -85,B 0,C 180,E1 -9511.874,E2 -9511.874} C_VEL
LIN {X 0,Y 432.38,Z 225.626,A -85,B 0,C 180,E1 -9515.538,E2 -9515.538} C_VEL
LIN {X 0,Y 432.351,Z 225.625,A -85,B 0,C 180,E1 -9519.046,E2 -9519.046} C_VEL
LIN {X 0,Y 432.362,Z 225.624,A -85,B 0,C 180,E1 -9522.01,E2 -9522.01} C_VEL
LIN {X 0,Y 432.397,Z 225.62,A -85,B 0,C 180,E1 -9524.927,E2 -9524.927} C_VEL
LIN {X 0,Y 432.46,Z 225.61,A -85,B 0,C 180,E1 -9527.803,E2 -9527.803} C_VEL
LIN {X 0,Y 432.493,Z 225.61,A -85,B 0,C 180,E1 -9531.59,E2 -9531.59} C_VEL
LIN {X 0,Y 432.598,Z 225.593,A -85,B 0,C 180,E1 -9534.406,E2 -9534.406} C_VEL
LIN {X 0,Y 432.601,Z 225.59,A -85,B 0,C 180,E1 -9538.138,E2 -9538.138} C_VEL
LIN {X 0,Y 432.731,Z 225.579,A -85,B 0,C 180,E1 -9540,E2 -9540} C_VEL
LIN {X 0,Y 432.585,Z 225.594,A -85,B 0,C 180,E1 -9542.794,E2 -9542.794} C_VEL
LIN {X 0,Y 432.543,Z 225.601,A -85,B 0,C 180,E1 -9546.488,E2 -9546.488} C_VEL
LIN {X 0,Y 432.44,Z 225.616,A -85,B 0,C 180,E1 -9549.353,E2 -9549.353} C_VEL
LIN {X 0,Y 432.432,Z 225.614,A -85,B 0,C 180,E1 -9552.803,E2 -9552.803} C_VEL
LIN {X 0,Y 432.413,Z 225.617,A -85,B 0,C 180,E1 -9556.478,E2 -9556.478} C_VEL
LIN {X 0,Y 432.339,Z 225.628,A -85,B 0,C 180,E1 -9559.961,E2 -9559.961} C_VEL
LIN {X 0,Y 432.318,Z 225.626,A -85,B 0,C 180,E1 -9562.964,E2 -9562.964} C_VEL
LIN {X 0,Y 432.351,Z 225.622,A -85,B 0,C 180,E1 -9566.034,E2 -9566.034} C_VEL
LIN {X 0,Y 432.344,Z 225.632,A -85,B 0,C 180,E1 -9569.188,E2 -9569.188} C_VEL
LIN {X 0,Y 432.325,Z 225.629,A -85,B 0,C 180,E1 -9572.443,E2 -9572.443} C_VEL
LIN {X 0,Y 432.345,Z 225.629,A -85,B 0,C 180,E1 -9575.632,E2 -9575.632} C_VEL
LIN {X 0,Y 432.339,Z 225.628,A -85,B 0,C 180,E1 -9578.714,E2 -9578.714} C_VEL
LIN {X 0,Y 432.326,Z 225.633,A -85,B 0,C 180,E1 -9581.798,E2 -9581.798} C_VEL
LIN {X 0,Y 432.335,Z 225.629,A -85,B 0,C 180,E1 -9584.348,E2 -9584.348} C_VEL
LIN {X 0,Y 432.318,Z 225.629,A -85,B 0,C 180,E1 -9587.016,E2 -9587.016} C_VEL
LIN {X 0,Y 432.315,Z 225.633,A -85,B 0,C 180,E1 -9589.824,E2 -9589.824} C_VEL
LIN {X 0,Y 432.308,Z 225.639,A -85,B 0,C 180,E1 -9593.022,E2 -9593.022} C_VEL
LIN {X 0,Y 432.36,Z 225.629,A -85,B 0,C 180,E1 -9595.997,E2 -9595.997} C_VEL
LIN {X 0,Y 432.349,Z 225.628,A -85,B 0,C 180,E1 -9599.49,E2 -9599.49} C_VEL
LIN {X 0,Y 432.412,Z 225.699,A -85,B 0,C 180,E1 -9601.051,E2 -9601.051} C_VEL
LIN {X 0,Y 434.223,Z 235.45,A -85,B 0,C 180,E1 -9603.311,E2 -9603.311} C_VEL
LIN {X 0,Y 434.082,Z 243.794,A -85,B 0,C 180,E1 -9605.105,E2 -9605.105} C_VEL
LIN {X 0,Y 434.032,Z 245.146,A -85,B 0,C 180,E1 -9605.39,E2 -9605.39} C_VEL
LIN {X 0,Y 438.084,Z 264.535,A -85,B 0,C 180,E1 -9605.922,E2 -9605.922} C_VEL
LIN {X 0,Y 436.981,Z 352.219,A -85,B 0,C 180,E1 -9607.388,E2 -9607.388} C_VEL
LIN {X 0,Y 436.634,Z 364.96,A -85,B 0,C 180,E1 -9607.774,E2 -9607.774} C_VEL
LIN {X 0,Y 436.117,Z 378.044,A -85,B 0,C 180,E1 -9608.369,E2 -9608.369} C_VEL
LIN {X 0,Y 435.53,Z 389.586,A -85,B 0,C 180,E1 -9609.082,E2 -9609.082} C_VEL
LIN {X 0,Y 434.835,Z 401.04,A -85,B 0,C 180,E1 -9610.003,E2 -9610.003} C_VEL
LIN {X 0,Y 434.126,Z 410.873,A -85,B 0,C 180,E1 -9610.986,E2 -9610.986} C_VEL
LIN {X 0,Y 433.538,Z 419.664,A -85,B 0,C 180,E1 -9612.061,E2 -9612.061} C_VEL
LIN {X 0,Y 433.028,Z 426.865,A -85,B 0,C 180,E1 -9613.118,E2 -9613.118} C_VEL
LIN {X 0,Y 432.12,Z 430.586,A -85,B 0,C 180,E1 -9613.717,E2 -9613.717} C_VEL
LIN {X 0,Y 428.865,Z 436.235,A -85,B 0,C 180,E1 -9614.713,E2 -9614.713} C_VEL
LIN {X 0,Y 425.659,Z 441.285,A -85,B 0,C 180,E1 -9615.778,E2 -9615.778} C_VEL
LIN {X 0,Y 424.836,Z 443.932,A -85,B 0,C 180,E1 -9616.476,E2 -9616.476} C_VEL
LIN {X 0,Y 424.51,Z 448.844,A -85,B 0,C 180,E1 -9618.068,E2 -9618.068} C_VEL
LIN {X 0,Y 424.259,Z 452.134,A -85,B 0,C 180,E1 -9619.501,E2 -9619.501} C_VEL
LIN {X 0,Y 424.105,Z 455.013,A -85,B 0,C 180,E1 -9621.423,E2 -9621.423} C_VEL
LIN {X 0,Y 424.11,Z 455.834,A -85,B 0,C 180,E1 -9622.382,E2 -9622.382} C_VEL
LIN {X 0,Y 424.168,Z 456.298,A -85,B 0,C 180,E1 -9623.795,E2 -9623.795} C_VEL
LIN {X 0,Y 424.133,Z 455.862,A -85,B 0,C 180,E1 -9625.247,E2 -9625.247} C_VEL
LIN {X 0,Y 424.085,Z 455.094,A -85,B 0,C 180,E1 -9626.199,E2 -9626.199} C_VEL
LIN {X 0,Y 424.184,Z 453.887,A -85,B 0,C 180,E1 -9627.151,E2 -9627.151} C_VEL
LIN {X 0,Y 424.234,Z 451.337,A -85,B 0,C 180,E1 -9628.576,E2 -9628.576} C_VEL
LIN {X 0,Y 424.339,Z 447.794,A -85,B 0,C 180,E1 -9630,E2 -9630} C_VEL
LIN {X 0,Y 424.554,Z 443.154,A -85,B 0,C 180,E1 -9631.423,E2 -9631.423} C_VEL
LIN {X 0,Y 424.871,Z 437.284,A -85,B 0,C 180,E1 -9632.844,E2 -9632.844} C_VEL
LIN {X 0,Y 425.349,Z 429.974,A -85,B 0,C 180,E1 -9634.264,E2 -9634.264} C_VEL
LIN {X 0,Y 426.032,Z 420.894,A -85,B 0,C 180,E1 -9635.68,E2 -9635.68} C_VEL
LIN {X 0,Y 426.721,Z 410.412,A -85,B 0,C 180,E1 -9636.977,E2 -9636.977} C_VEL
LIN {X 0,Y 427.421,Z 399.742,A -85,B 0,C 180,E1 -9638.034,E2 -9638.034} C_VEL
LIN {X 0,Y 427.982,Z 389.39,A -85,B 0,C 180,E1 -9638.856,E2 -9638.856} C_VEL
LIN {X 0,Y 428.571,Z 376.956,A -85,B 0,C 180,E1 -9639.617,E2 -9639.617} C_VEL
LIN {X 0,Y 429.054,Z 363.831,A -85,B 0,C 180,E1 -9640.202,E2 -9640.202} C_VEL
LIN {X 0,Y 429.287,Z 352.14,A -85,B 0,C 180,E1 -9640.55,E2 -9640.55} C_VEL
LIN {X 0,Y 430.235,Z 264.712,A -85,B 0,C 180,E1 -9642.021,E2 -9642.021} C_VEL
LIN {X 0,Y 426.708,Z 245.154,A -85,B 0,C 180,E1 -9642.514,E2 -9642.514} C_VEL
LIN {X 0,Y 427.002,Z 235.705,A -85,B 0,C 180,E1 -9644.537,E2 -9644.537} C_VEL
LIN {X 0,Y 425.369,Z 226.503,A -85,B 0,C 180,E1 -9646.654,E2 -9646.654} C_VEL
LIN {X 0,Y 425.331,Z 226.501,A -85,B 0,C 180,E1 -9649.635,E2 -9649.635} C_VEL
LIN {X 0,Y 425.291,Z 226.508,A -85,B 0,C 180,E1 -9652.339,E2 -9652.339} C_VEL
LIN {X 0,Y 425.324,Z 226.508,A -85,B 0,C 180,E1 -9654.657,E2 -9654.657} C_VEL
LIN {X 0,Y 425.302,Z 226.503,A -85,B 0,C 180,E1 -9657.561,E2 -9657.561} C_VEL
LIN {X 0,Y 425.29,Z 226.511,A -85,B 0,C 180,E1 -9660.816,E2 -9660.816} C_VEL
LIN {X 0,Y 425.314,Z 226.505,A -85,B 0,C 180,E1 -9664.288,E2 -9664.288} C_VEL
LIN {X 0,Y 425.28,Z 226.506,A -85,B 0,C 180,E1 -9667.694,E2 -9667.694} C_VEL
LIN {X 0,Y 425.282,Z 226.511,A -85,B 0,C 180,E1 -9670.52,E2 -9670.52} C_VEL
LIN {X 0,Y 425.259,Z 226.509,A -85,B 0,C 180,E1 -9673.351,E2 -9673.351} C_VEL
LIN {X 0,Y 425.257,Z 226.516,A -85,B 0,C 180,E1 -9676.649,E2 -9676.649} C_VEL
LIN {X 0,Y 425.285,Z 226.506,A -85,B 0,C 180,E1 -9679.872,E2 -9679.872} C_VEL
LIN {X 0,Y 425.278,Z 226.512,A -85,B 0,C 180,E1 -9682.489,E2 -9682.489} C_VEL
LIN {X 0,Y 425.308,Z 226.503,A -85,B 0,C 180,E1 -9685.817,E2 -9685.817} C_VEL
LIN {X 0,Y 425.292,Z 226.506,A -85,B 0,C 180,E1 -9689.239,E2 -9689.239} C_VEL
LIN {X 0,Y 425.346,Z 226.503,A -85,B 0,C 180,E1 -9692.442,E2 -9692.442} C_VEL
LIN {X 0,Y 425.346,Z 226.498,A -85,B 0,C 180,E1 -9695.602,E2 -9695.602} C_VEL
LIN {X 0,Y 425.294,Z 226.511,A -85,B 0,C 180,E1 -9698.681,E2 -9698.681} C_VEL
LIN {X 0,Y 425.322,Z 226.501,A -85,B 0,C 180,E1 -9701.702,E2 -9701.702} C_VEL
LIN {X 0,Y 425.348,Z 226.505,A -85,B 0,C 180,E1 -9704.67,E2 -9704.67} C_VEL
LIN {X 0,Y 425.413,Z 226.489,A -85,B 0,C 180,E1 -9707.598,E2 -9707.598} C_VEL
LIN {X 0,Y 425.408,Z 226.49,A -85,B 0,C 180,E1 -9711.449,E2 -9711.449} C_VEL
LIN {X 0,Y 425.542,Z 226.477,A -85,B 0,C 180,E1 -9714.313,E2 -9714.313} C_VEL
LIN {X 0,Y 425.574,Z 226.471,A -85,B 0,C 180,E1 -9718.107,E2 -9718.107} C_VEL
LIN {X 0,Y 425.7,Z 226.455,A -85,B 0,C 180,E1 -9720,E2 -9720} C_VEL
LIN {X 0,Y 425.538,Z 226.478,A -85,B 0,C 180,E1 -9722.84,E2 -9722.84} C_VEL
LIN {X 0,Y 425.531,Z 226.482,A -85,B 0,C 180,E1 -9726.639,E2 -9726.639} C_VEL
LIN {X 0,Y 425.4,Z 226.491,A -85,B 0,C 180,E1 -9729.509,E2 -9729.509} C_VEL
LIN {X 0,Y 425.394,Z 226.495,A -85,B 0,C 180,E1 -9732.904,E2 -9732.904} C_VEL
LIN {X 0,Y 425.361,Z 226.503,A -85,B 0,C 180,E1 -9736.605,E2 -9736.605} C_VEL
LIN {X 0,Y 425.329,Z 226.5,A -85,B 0,C 180,E1 -9739.635,E2 -9739.635} C_VEL
LIN {X 0,Y 425.288,Z 226.509,A -85,B 0,C 180,E1 -9742.339,E2 -9742.339} C_VEL
LIN {X 0,Y 425.321,Z 226.507,A -85,B 0,C 180,E1 -9744.657,E2 -9744.657} C_VEL
LIN {X 0,Y 425.272,Z 226.507,A -85,B 0,C 180,E1 -9747.563,E2 -9747.563} C_VEL
LIN {X 0,Y 425.29,Z 226.51,A -85,B 0,C 180,E1 -9750.761,E2 -9750.761} C_VEL
LIN {X 0,Y 425.31,Z 226.506,A -85,B 0,C 180,E1 -9754.288,E2 -9754.288} C_VEL
LIN {X 0,Y 425.276,Z 226.506,A -85,B 0,C 180,E1 -9757.695,E2 -9757.695} C_VEL
LIN {X 0,Y 425.266,Z 226.515,A -85,B 0,C 180,E1 -9760.518,E2 -9760.518} C_VEL
LIN {X 0,Y 425.255,Z 226.509,A -85,B 0,C 180,E1 -9763.351,E2 -9763.351} C_VEL
LIN {X 0,Y 425.261,Z 226.51,A -85,B 0,C 180,E1 -9766.044,E2 -9766.044} C_VEL
LIN {X 0,Y 425.277,Z 226.506,A -85,B 0,C 180,E1 -9769.48,E2 -9769.48} C_VEL
LIN {X 0,Y 425.277,Z 226.513,A -85,B 0,C 180,E1 -9772.489,E2 -9772.489} C_VEL
LIN {X 0,Y 425.308,Z 226.503,A -85,B 0,C 180,E1 -9775.817,E2 -9775.817} C_VEL
LIN {X 0,Y 425.292,Z 226.508,A -85,B 0,C 180,E1 -9779.239,E2 -9779.239} C_VEL
LIN {X 0,Y 425.347,Z 226.505,A -85,B 0,C 180,E1 -9782.442,E2 -9782.442} C_VEL
LIN {X 0,Y 425.351,Z 226.508,A -85,B 0,C 180,E1 -9783.379,E2 -9783.379} C_VEL
LIN {X 0,Y 427.702,Z 238.912,A -85,B 0,C 180,E1 -9786.003,E2 -9786.003} C_VEL
LIN {X 0,Y 427.645,Z 244.467,A -85,B 0,C 180,E1 -9787.104,E2 -9787.104} C_VEL
LIN {X 0,Y 426.67,Z 262.041,A -85,B 0,C 180,E1 -9790.517,E2 -9790.517} C_VEL
LIN {X 0,Y 426.37,Z 267.229,A -85,B 0,C 180,E1 -9791.516,E2 -9791.516} C_VEL
LIN {X 0,Y 429.975,Z 291.996,A -85,B 0,C 180,E1 -9792.083,E2 -9792.083} C_VEL
LIN {X 0,Y 429.192,Z 375.695,A -85,B 0,C 180,E1 -9793.501,E2 -9793.501} C_VEL
LIN {X 0,Y 428.674,Z 388.917,A -85,B 0,C 180,E1 -9793.908,E2 -9793.908} C_VEL
LIN {X 0,Y 428.153,Z 401.079,A -85,B 0,C 180,E1 -9794.469,E2 -9794.469} C_VEL
LIN {X 0,Y 427.507,Z 413.338,A -85,B 0,C 180,E1 -9795.238,E2 -9795.238} C_VEL
LIN {X 0,Y 426.768,Z 425.272,A -85,B 0,C 180,E1 -9796.216,E2 -9796.216} C_VEL
LIN {X 0,Y 426.19,Z 435.402,A -85,B 0,C 180,E1 -9797.258,E2 -9797.258} C_VEL
LIN {X 0,Y 425.681,Z 443.941,A -85,B 0,C 180,E1 -9798.332,E2 -9798.332} C_VEL
LIN {X 0,Y 425.048,Z 453.178,A -85,B 0,C 180,E1 -9799.761,E2 -9799.761} C_VEL
LIN {X 0,Y 424.679,Z 460.608,A -85,B 0,C 180,E1 -9801.195,E2 -9801.195} C_VEL
LIN {X 0,Y 424.344,Z 467.431,A -85,B 0,C 180,E1 -9802.865,E2 -9802.865} C_VEL
LIN {X 0,Y 424.189,Z 471.927,A -85,B 0,C 180,E1 -9804.295,E2 -9804.295} C_VEL
LIN {X 0,Y 424.199,Z 474.299,A -85,B 0,C 180,E1 -9805.248,E2 -9805.248} C_VEL
LIN {X 0,Y 424.099,Z 476.234,A -85,B 0,C 180,E1 -9806.199,E2 -9806.199} C_VEL
LIN {X 0,Y 424.132,Z 477.747,A -85,B 0,C 180,E1 -9807.151,E2 -9807.151} C_VEL
LIN {X 0,Y 424.129,Z 478.806,A -85,B 0,C 180,E1 -9808.101,E2 -9808.101} C_VEL
LIN {X 0,Y 424.085,Z 479.751,A -85,B 0,C 180,E1 -9810,E2 -9810} C_VEL
LIN {X 0,Y 424.088,Z 479.64,A -85,B 0,C 180,E1 -9810.95,E2 -9810.95} C_VEL
LIN {X 0,Y 424.129,Z 479.097,A -85,B 0,C 180,E1 -9811.899,E2 -9811.899} C_VEL
LIN {X 0,Y 424.13,Z 478.16,A -85,B 0,C 180,E1 -9812.849,E2 -9812.849} C_VEL
LIN {X 0,Y 424.097,Z 476.829,A -85,B 0,C 180,E1 -9813.801,E2 -9813.801} C_VEL
LIN {X 0,Y 424.206,Z 474.021,A -85,B 0,C 180,E1 -9815.228,E2 -9815.228} C_VEL
LIN {X 0,Y 424.301,Z 470.193,A -85,B 0,C 180,E1 -9816.658,E2 -9816.658} C_VEL
LIN {X 0,Y 424.547,Z 465.251,A -85,B 0,C 180,E1 -9818.089,E2 -9818.089} C_VEL
LIN {X 0,Y 424.947,Z 459.045,A -85,B 0,C 180,E1 -9819.52,E2 -9819.52} C_VEL
LIN {X 0,Y 425.442,Z 451.319,A -85,B 0,C 180,E1 -9820.951,E2 -9820.951} C_VEL
LIN {X 0,Y 426.271,Z 441.651,A -85,B 0,C 180,E1 -9822.376,E2 -9822.376} C_VEL
LIN {X 0,Y 426.989,Z 432.361,A -85,B 0,C 180,E1 -9823.488,E2 -9823.488} C_VEL
LIN {X 0,Y 427.618,Z 421.852,A -85,B 0,C 180,E1 -9824.515,E2 -9824.515} C_VEL
LIN {X 0,Y 428.472,Z 409.42,A -85,B 0,C 180,E1 -9825.459,E2 -9825.459} C_VEL
LIN {X 0,Y 429.241,Z 397.218,A -85,B 0,C 180,E1 -9826.161,E2 -9826.161} C_VEL
LIN {X 0,Y 429.804,Z 385.312,A -85,B 0,C 180,E1 -9826.658,E2 -9826.658} C_VEL
LIN {X 0,Y 430.208,Z 372.325,A -85,B 0,C 180,E1 -9827.009,E2 -9827.009} C_VEL
LIN {X 0,Y 430.967,Z 290.784,A -85,B 0,C 180,E1 -9828.397,E2 -9828.397} C_VEL
LIN {X 0,Y 426.843,Z 266.964,A -85,B 0,C 180,E1 -9829.043,E2 -9829.043} C_VEL
LIN {X 0,Y 427.992,Z 249.691,A -85,B 0,C 180,E1 -9832.443,E2 -9832.443} C_VEL
LIN {X 0,Y 428.397,Z 242.135,A -85,B 0,C 180,E1 -9833.956,E2 -9833.956} C_VEL
LIN {X 0,Y 426.499,Z 232.067,A -85,B 0,C 180,E1 -9836.155,E2 -9836.155} C_VEL
LIN {X 0,Y 425.355,Z 226.506,A -85,B 0,C 180,E1 -9837.417,E2 -9837.417} C_VEL
LIN {X 0,Y 425.289,Z 226.509,A -85,B 0,C 180,E1 -9840.816,E2 -9840.816} C_VEL
LIN {X 0,Y 425.312,Z 226.504,A -85,B 0,C 180,E1 -9844.288,E2 -9844.288} C_VEL
LIN {X 0,Y 425.278,Z 226.513,A -85,B 0,C 180,E1 -9847.694,E2 -9847.694} C_VEL
LIN {X 0,Y 425.277,Z 226.508,A -85,B 0,C 180,E1 -9850.52,E2 -9850.52} C_VEL
LIN {X 0,Y 425.261,Z 226.512,A -85,B 0,C 180,E1 -9853.956,E2 -9853.956} C_VEL
LIN {X 0,Y 425.271,Z 226.514,A -85,B 0,C 180,E1 -9857.346,E2 -9857.346} C_VEL
LIN {X 0,Y 425.266,Z 226.511,A -85,B 0,C 180,E1 -9859.87,E2 -9859.87} C_VEL
LIN {X 0,Y 425.276,Z 226.506,A -85,B 0,C 180,E1 -9862.489,E2 -9862.489} C_VEL
LIN {X 0,Y 425.306,Z 226.503,A -85,B 0,C 180,E1 -9865.817,E2 -9865.817} C_VEL
LIN {X 0,Y 425.291,Z 226.51,A -85,B 0,C 180,E1 -9869.239,E2 -9869.239} C_VEL
LIN {X 0,Y 425.3,Z 226.504,A -85,B 0,C 180,E1 -9872.439,E2 -9872.439} C_VEL
LIN {X 0,Y 425.348,Z 226.503,A -85,B 0,C 180,E1 -9875.602,E2 -9875.602} C_VEL
LIN {X 0,Y 425.294,Z 226.502,A -85,B 0,C 180,E1 -9878.682,E2 -9878.682} C_VEL
LIN {X 0,Y 425.323,Z 226.504,A -85,B 0,C 180,E1 -9881.702,E2 -9881.702} C_VEL
LIN {X 0,Y 425.35,Z 226.497,A -85,B 0,C 180,E1 -9884.671,E2 -9884.671} C_VEL
LIN {X 0,Y 425.413,Z 226.489,A -85,B 0,C 180,E1 -9887.598,E2 -9887.598} C_VEL
LIN {X 0,Y 425.443,Z 226.49,A -85,B 0,C 180,E1 -9891.45,E2 -9891.45} C_VEL
LIN {X 0,Y 425.554,Z 226.471,A -85,B 0,C 180,E1 -9894.313,E2 -9894.313} C_VEL
LIN {X 0,Y 425.571,Z 226.466,A -85,B 0,C 180,E1 -9898.107,E2 -9898.107} C_VEL
LIN {X 0,Y 425.7,Z 226.455,A -85,B 0,C 180,E1 -9900,E2 -9900} C_VEL
LIN {X 0,Y 425.539,Z 226.472,A -85,B 0,C 180,E1 -9902.84,E2 -9902.84} C_VEL
LIN {X 0,Y 425.499,Z 226.479,A -85,B 0,C 180,E1 -9906.488,E2 -9906.488} C_VEL
LIN {X 0,Y 425.399,Z 226.495,A -85,B 0,C 180,E1 -9909.51,E2 -9909.51} C_VEL
LIN {X 0,Y 425.395,Z 226.492,A -85,B 0,C 180,E1 -9912.904,E2 -9912.904} C_VEL
LIN {X 0,Y 425.362,Z 226.496,A -85,B 0,C 180,E1 -9916.605,E2 -9916.605} C_VEL
LIN {X 0,Y 425.329,Z 226.504,A -85,B 0,C 180,E1 -9919.636,E2 -9919.636} C_VEL
LIN {X 0,Y 425.305,Z 226.504,A -85,B 0,C 180,E1 -9923.365,E2 -9923.365} C_VEL
LIN {X 0,Y 425.341,Z 226.496,A -85,B 0,C 180,E1 -9926.842,E2 -9926.842} C_VEL
LIN {X 0,Y 425.292,Z 226.506,A -85,B 0,C 180,E1 -9929.72,E2 -9929.72} C_VEL
LIN {X 0,Y 425.284,Z 226.51,A -85,B 0,C 180,E1 -9933.048,E2 -9933.048} C_VEL
LIN {X 0,Y 425.283,Z 226.506,A -85,B 0,C 180,E1 -9935.929,E2 -9935.929} C_VEL
LIN {X 0,Y 425.282,Z 226.51,A -85,B 0,C 180,E1 -9939.041,E2 -9939.041} C_VEL
LIN {X 0,Y 425.284,Z 226.509,A -85,B 0,C 180,E1 -9941.957,E2 -9941.957} C_VEL
LIN {X 0,Y 425.286,Z 226.513,A -85,B 0,C 180,E1 -9945.283,E2 -9945.283} C_VEL
LIN {X 0,Y 425.267,Z 226.513,A -85,B 0,C 180,E1 -9948.62,E2 -9948.62} C_VEL
LIN {X 0,Y 425.283,Z 226.511,A -85,B 0,C 180,E1 -9951.1,E2 -9951.1} C_VEL
LIN {X 0,Y 425.3,Z 226.509,A -85,B 0,C 180,E1 -9954.664,E2 -9954.664} C_VEL
LIN {X 0,Y 425.267,Z 226.51,A -85,B 0,C 180,E1 -9958.073,E2 -9958.073} C_VEL
LIN {X 0,Y 425.359,Z 226.688,A -85,B 0,C 180,E1 -9960.799,E2 -9960.799} C_VEL
LIN {X 0,Y 427.272,Z 236.586,A -85,B 0,C 180,E1 -9963.135,E2 -9963.135} C_VEL
LIN {X 0,Y 427.284,Z 242.436,A -85,B 0,C 180,E1 -9964.421,E2 -9964.421} C_VEL
LIN {X 0,Y 427.167,Z 245.248,A -85,B 0,C 180,E1 -9965.027,E2 -9965.027} C_VEL
LIN {X 0,Y 431.384,Z 265.11,A -85,B 0,C 180,E1 -9965.605,E2 -9965.605} C_VEL
LIN {X 0,Y 430.259,Z 353.216,A -85,B 0,C 180,E1 -9967.11,E2 -9967.11} C_VEL
LIN {X 0,Y 429.856,Z 366.457,A -85,B 0,C 180,E1 -9967.532,E2 -9967.532} C_VEL
LIN {X 0,Y 429.328,Z 379.194,A -85,B 0,C 180,E1 -9968.135,E2 -9968.135} C_VEL
LIN {X 0,Y 428.707,Z 390.458,A -85,B 0,C 180,E1 -9968.859,E2 -9968.859} C_VEL
LIN {X 0,Y 427.948,Z 402.13,A -85,B 0,C 180,E1 -9969.826,E2 -9969.826} C_VEL
LIN {X 0,Y 427.139,Z 412.599,A -85,B 0,C 180,E1 -9970.912,E2 -9970.912} C_VEL
LIN {X 0,Y 426.531,Z 421.125,A -85,B 0,C 180,E1 -9972.004,E2 -9972.004} C_VEL
LIN {X 0,Y 425.89,Z 429.379,A -85,B 0,C 180,E1 -9973.293,E2 -9973.293} C_VEL
LIN {X 0,Y 425.312,Z 436.564,A -85,B 0,C 180,E1 -9974.669,E2 -9974.669} C_VEL
LIN {X 0,Y 424.909,Z 442.662,A -85,B 0,C 180,E1 -9976.123,E2 -9976.123} C_VEL
LIN {X 0,Y 424.836,Z 443.932,A -85,B 0,C 180,E1 -9976.476,E2 -9976.476} C_VEL
LIN {X 0,Y 424.027,Z 446.422,A -85,B 0,C 180,E1 -9977.193,E2 -9977.193} C_VEL
LIN {X 0,Y 420.901,Z 449.999,A -85,B 0,C 180,E1 -9978.376,E2 -9978.376} C_VEL
LIN {X 0,Y 417.801,Z 452.771,A -85,B 0,C 180,E1 -9979.613,E2 -9979.613} C_VEL
LIN {X 0,Y 417.05,Z 454.001,A -85,B 0,C 180,E1 -9980.402,E2 -9980.402} C_VEL
LIN {X 0,Y 417.033,Z 455.988,A -85,B 0,C 180,E1 -9982.252,E2 -9982.252} C_VEL
LIN {X 0,Y 417.095,Z 456.497,A -85,B 0,C 180,E1 -9983.799,E2 -9983.799} C_VEL
LIN {X 0,Y 417.038,Z 456.094,A -85,B 0,C 180,E1 -9985.166,E2 -9985.166} C_VEL
LIN {X 0,Y 416.998,Z 455.362,A -85,B 0,C 180,E1 -9986.134,E2 -9986.134} C_VEL
LIN {X 0,Y 417.079,Z 454.19,A -85,B 0,C 180,E1 -9987.102,E2 -9987.102} C_VEL
LIN {X 0,Y 417.131,Z 452.613,A -85,B 0,C 180,E1 -9988.069,E2 -9988.069} C_VEL
LIN {X 0,Y 417.235,Z 449.454,A -85,B 0,C 180,E1 -9989.517,E2 -9989.517} C_VEL
LIN {X 0,Y 417.383,Z 445.248,A -85,B 0,C 180,E1 -9990.965,E2 -9990.965} C_VEL
LIN {X 0,Y 417.843,Z 438.866,A -85,B 0,C 180,E1 -9992.651,E2 -9992.651} C_VEL
LIN {X 0,Y 418.176,Z 431.907,A -85,B 0,C 180,E1 -9994.096,E2 -9994.096} C_VEL
LIN {X 0,Y 418.888,Z 423.192,A -85,B 0,C 180,E1 -9995.536,E2 -9995.536} C_VEL
LIN {X 0,Y 419.571,Z 414.276,A -85,B 0,C 180,E1 -9996.734,E2 -9996.734} C_VEL
LIN {X 0,Y 420.2,Z 404.484,A -85,B 0,C 180,E1 -9997.81,E2 -9997.81} C_VEL
LIN {X 0,Y 420.839,Z 393.647,A -85,B 0,C 180,E1 -9998.765,E2 -9998.765} C_VEL
LIN {X 0,Y 421.47,Z 381.517,A -85,B 0,C 180,E1 -9999.599,E2 -9999.599} C_VEL
LIN {X 0,Y 422.015,Z 368.77,A -85,B 0,C 180,E1 -10000.252,E2 -10000.252} C_VEL
LIN {X 0,Y 422.314,Z 355.526,A -85,B 0,C 180,E1 -10000.711,E2 -10000.711} C_VEL
LIN {X 0,Y 422.68,Z 335.777,A -85,B 0,C 180,E1 -10001.089,E2 -10001.089} C_VEL
LIN {X 0,Y 423.338,Z 265.062,A -85,B 0,C 180,E1 -10002.288,E2 -10002.288} C_VEL
LIN {X 0,Y 419.771,Z 245.381,A -85,B 0,C 180,E1 -10002.786,E2 -10002.786} C_VEL
LIN {X 0,Y 419.97,Z 236.203,A -85,B 0,C 180,E1 -10004.785,E2 -10004.785} C_VEL
LIN {X 0,Y 418.339,Z 227.378,A -85,B 0,C 180,E1 -10006.86,E2 -10006.86} C_VEL
LIN {X 0,Y 418.274,Z 227.38,A -85,B 0,C 180,E1 -10009.79,E2 -10009.79} C_VEL
LIN {X 0,Y 418.235,Z 227.391,A -85,B 0,C 180,E1 -10012.736,E2 -10012.736} C_VEL
LIN {X 0,Y 418.24,Z 227.383,A -85,B 0,C 180,E1 -10015.906,E2 -10015.906} C_VEL
LIN {X 0,Y 418.263,Z 227.382,A -85,B 0,C 180,E1 -10019.162,E2 -10019.162} C_VEL
LIN {X 0,Y 418.26,Z 227.386,A -85,B 0,C 180,E1 -10022.844,E2 -10022.844} C_VEL
LIN {X 0,Y 418.247,Z 227.384,A -85,B 0,C 180,E1 -10026.238,E2 -10026.238} C_VEL
LIN {X 0,Y 418.248,Z 227.382,A -85,B 0,C 180,E1 -10029.682,E2 -10029.682} C_VEL
LIN {X 0,Y 418.231,Z 227.387,A -85,B 0,C 180,E1 -10032.321,E2 -10032.321} C_VEL
LIN {X 0,Y 418.237,Z 227.386,A -85,B 0,C 180,E1 -10035.108,E2 -10035.108} C_VEL
LIN {X 0,Y 418.235,Z 227.383,A -85,B 0,C 180,E1 -10037.766,E2 -10037.766} C_VEL
LIN {X 0,Y 418.246,Z 227.389,A -85,B 0,C 180,E1 -10040.62,E2 -10040.62} C_VEL
LIN {X 0,Y 418.243,Z 227.383,A -85,B 0,C 180,E1 -10043.975,E2 -10043.975} C_VEL
LIN {X 0,Y 418.259,Z 227.382,A -85,B 0,C 180,E1 -10047.156,E2 -10047.156} C_VEL
LIN {X 0,Y 418.27,Z 227.384,A -85,B 0,C 180,E1 -10050.895,E2 -10050.895} C_VEL
LIN {X 0,Y 418.262,Z 227.382,A -85,B 0,C 180,E1 -10054.095,E2 -10054.095} C_VEL
LIN {X 0,Y 418.238,Z 227.384,A -85,B 0,C 180,E1 -10057.264,E2 -10057.264} C_VEL
LIN {X 0,Y 418.284,Z 227.382,A -85,B 0,C 180,E1 -10060.364,E2 -10060.364} C_VEL
LIN {X 0,Y 418.317,Z 227.374,A -85,B 0,C 180,E1 -10063.404,E2 -10063.404} C_VEL
LIN {X 0,Y 418.347,Z 227.373,A -85,B 0,C 180,E1 -10066.999,E2 -10066.999} C_VEL
LIN {X 0,Y 418.339,Z 227.374,A -85,B 0,C 180,E1 -10070.328,E2 -10070.328} C_VEL
LIN {X 0,Y 418.461,Z 227.356,A -85,B 0,C 180,E1 -10073.248,E2 -10073.248} C_VEL
LIN {X 0,Y 418.335,Z 227.372,A -85,B 0,C 180,E1 -10075.181,E2 -10075.181} C_VEL
LIN {X 0,Y 418.543,Z 227.347,A -85,B 0,C 180,E1 -10078.075,E2 -10078.075} C_VEL
LIN {X 0,Y 418.669,Z 227.331,A -85,B 0,C 180,E1 -10080,E2 -10080} C_VEL
LIN {X 0,Y 418.494,Z 227.355,A -85,B 0,C 180,E1 -10082.888,E2 -10082.888} C_VEL
LIN {X 0,Y 418.494,Z 227.357,A -85,B 0,C 180,E1 -10086.751,E2 -10086.751} C_VEL
LIN {X 0,Y 418.4,Z 227.369,A -85,B 0,C 180,E1 -10088.695,E2 -10088.695} C_VEL
LIN {X 0,Y 418.356,Z 227.376,A -85,B 0,C 180,E1 -10092.614,E2 -10092.614} C_VEL
LIN {X 0,Y 418.303,Z 227.375,A -85,B 0,C 180,E1 -10095.594,E2 -10095.594} C_VEL
LIN {X 0,Y 418.277,Z 227.386,A -85,B 0,C 180,E1 -10098.617,E2 -10098.617} C_VEL
LIN {X 0,Y 418.234,Z 227.384,A -85,B 0,C 180,E1 -10101.696,E2 -10101.696} C_VEL
LIN {X 0,Y 418.268,Z 227.383,A -85,B 0,C 180,E1 -10104.86,E2 -10104.86} C_VEL
LIN {X 0,Y 418.248,Z 227.384,A -85,B 0,C 180,E1 -10108.066,E2 -10108.066} C_VEL
LIN {X 0,Y 418.211,Z 227.387,A -85,B 0,C 180,E1 -10111.396,E2 -10111.396} C_VEL
LIN {X 0,Y 418.264,Z 227.387,A -85,B 0,C 180,E1 -10114.58,E2 -10114.58} C_VEL
LIN {X 0,Y 418.222,Z 227.386,A -85,B 0,C 180,E1 -10117.832,E2 -10117.832} C_VEL
LIN {X 0,Y 418.217,Z 227.389,A -85,B 0,C 180,E1 -10120.949,E2 -10120.949} C_VEL
LIN {X 0,Y 418.208,Z 227.387,A -85,B 0,C 180,E1 -10123.729,E2 -10123.729} C_VEL
LIN {X 0,Y 418.208,Z 227.393,A -85,B 0,C 180,E1 -10126.449,E2 -10126.449} C_VEL
LIN {X 0,Y 418.221,Z 227.386,A -85,B 0,C 180,E1 -10129.131,E2 -10129.131} C_VEL
LIN {X 0,Y 418.226,Z 227.388,A -85,B 0,C 180,E1 -10132.167,E2 -10132.167} C_VEL
LIN {X 0,Y 418.266,Z 227.38,A -85,B 0,C 180,E1 -10135.42,E2 -10135.42} C_VEL
LIN {X 0,Y 418.213,Z 227.394,A -85,B 0,C 180,E1 -10138.604,E2 -10138.604} C_VEL
LIN {X 0,Y 418.291,Z 227.382,A -85,B 0,C 180,E1 -10141.937,E2 -10141.937} C_VEL
LIN {X 0,Y 418.345,Z 227.538,A -85,B 0,C 180,E1 -10143.195,E2 -10143.195} C_VEL
